LIN {X 70.213, Y 92.532, Z 255.75, A 0, B 90, C 0, E1 0, E2 0, E3 0, E4 0} C_DIS
LIN {X 73.181, Y 90.036, Z 255.75, A 0, B 90, C 0, E1 0, E2 0, E3 0, E4 0} C_DIS
LIN {X 75.725, Y 87.108, Z 255.75, A 0, B 90, C 0, E1 0, E2 0, E3 0, E4 0} C_DIS
LIN {X 77.888, Y 83.886, Z 255.75, A 0, B 90, C 0, E1 0, E2 0, E3 0, E4 0} C_DIS
LIN {X 79.733, Y 80.472, Z 255.75, A 0, B 90, C 0, E1 0, E2 0, E3 0, E4 0} C_DIS
LIN {X 81.33, Y 76.933, Z 255.75, A 0, B 90, C 0, E1 0, E2 0, E3 0, E4 0} C_DIS
LIN {X 82.75, Y 73.32, Z 255.75, A 0, B 90, C 0, E1 0, E2 0, E3 0, E4 0} C_DIS
LIN {X 84.078, Y 69.672, Z 255.75, A 0, B 90, C 0, E1 0, E2 0, E3 0, E4 0} C_DIS
LIN {X 85.426, Y 66.031, Z 255.75, A 0, B 90, C 0, E1 0, E2 0, E3 0, E4 0} C_DIS
LIN {X 86.966, Y 62.469, Z 255.75, A 0, B 90, C 0, E1 0, E2 0, E3 0, E4 0} C_DIS
LIN {X 88.949, Y 59.137, Z 255.75, A 0, B 90, C 0, E1 0, E2 0, E3 0, E4 0} C_DIS
LIN {X 91.538, Y 56.253, Z 255.75, A 0, B 90, C 0, E1 0, E2 0, E3 0, E4 0} C_DIS
LIN {X 94.581, Y 53.847, Z 255.75, A 0, B 90, C 0, E1 0, E2 0, E3 0, E4 0} C_DIS
LIN {X 97.829, Y 51.72, Z 255.75, A 0, B 90, C 0, E1 0, E2 0, E3 0, E4 0} C_DIS
LIN {X 101.131, Y 49.678, Z 255.75, A 0, B 90, C 0, E1 0, E2 0, E3 0, E4 0} C_DIS
LIN {X 104.407, Y 47.594, Z 255.75, A 0, B 90, C 0, E1 0, E2 0, E3 0, E4 0} C_DIS
LIN {X 107.602, Y 45.389, Z 255.75, A 0, B 90, C 0, E1 0, E2 0, E3 0, E4 0} C_DIS
LIN {X 110.666, Y 43.006, Z 255.75, A 0, B 90, C 0, E1 0, E2 0, E3 0, E4 0} C_DIS
LIN {X 113.544, Y 40.402, Z 255.75, A 0, B 90, C 0, E1 0, E2 0, E3 0, E4 0} C_DIS
LIN {X 116.164, Y 37.54, Z 255.75, A 0, B 90, C 0, E1 0, E2 0, E3 0, E4 0} C_DIS
LIN {X 118.433, Y 34.393, Z 255.75, A 0, B 90, C 0, E1 0, E2 0, E3 0, E4 0} C_DIS
LIN {X 120.224, Y 30.953, Z 255.75, A 0, B 90, C 0, E1 0, E2 0, E3 0, E4 0} C_DIS
LIN {X 121.382, Y 27.253, Z 255.75, A 0, B 90, C 0, E1 0, E2 0, E3 0, E4 0} C_DIS
LIN {X 121.779, Y 23.398, Z 255.75, A 0, B 90, C 0, E1 0, E2 0, E3 0, E4 0} C_DIS
LIN {X 121.393, Y 19.541, Z 255.75, A 0, B 90, C 0, E1 0, E2 0, E3 0, E4 0} C_DIS
LIN {X 120.325, Y 15.813, Z 255.75, A 0, B 90, C 0, E1 0, E2 0, E3 0, E4 0} C_DIS
LIN {X 118.73, Y 12.276, Z 255.75, A 0, B 90, C 0, E1 0, E2 0, E3 0, E4 0} C_DIS
LIN {X 116.749, Y 8.94, Z 255.75, A 0, B 90, C 0, E1 0, E2 0, E3 0, E4 0} C_DIS
LIN {X 114.484, Y 5.788, Z 255.75, A 0, B 90, C 0, E1 0, E2 0, E3 0, E4 0} C_DIS
LIN {X 112.003, Y 2.805, Z 255.75, A 0, B 90, C 0, E1 0, E2 0, E3 0, E4 0} C_DIS
LIN {X 109.464, Y 0, Z 255.75, A 0, B 90, C 0, E1 0, E2 0, E3 0, E4 0} C_DIS
LIN {X 106.746, Y -2.436, Z 255.75, A 0, B 90, C 0, E1 0, E2 0, E3 0, E4 0} C_DIS
LIN {X 104.005, Y -5.183, Z 255.75, A 0, B 90, C 0, E1 0, E2 0, E3 0, E4 0} C_DIS
LIN {X 101.28, Y -7.949, Z 255.75, A 0, B 90, C 0, E1 0, E2 0, E3 0, E4 0} C_DIS
LIN {X 98.625, Y -10.781, Z 255.75, A 0, B 90, C 0, E1 0, E2 0, E3 0, E4 0} C_DIS
LIN {X 96.18, Y -13.794, Z 255.75, A 0, B 90, C 0, E1 0, E2 0, E3 0, E4 0} C_DIS
LIN {X 94.209, Y -17.132, Z 255.75, A 0, B 90, C 0, E1 0, E2 0, E3 0, E4 0} C_DIS
LIN {X 93.035, Y -20.823, Z 255.75, A 0, B 90, C 0, E1 0, E2 0, E3 0, E4 0} C_DIS
LIN {X 92.662, Y -24.683, Z 255.75, A 0, B 90, C 0, E1 0, E2 0, E3 0, E4 0} C_DIS
LIN {X 92.802, Y -28.561, Z 255.75, A 0, B 90, C 0, E1 0, E2 0, E3 0, E4 0} C_DIS
LIN {X 93.225, Y -32.42, Z 255.75, A 0, B 90, C 0, E1 0, E2 0, E3 0, E4 0} C_DIS
LIN {X 93.804, Y -36.259, Z 255.75, A 0, B 90, C 0, E1 0, E2 0, E3 0, E4 0} C_DIS
LIN {X 94.463, Y -40.085, Z 255.75, A 0, B 90, C 0, E1 0, E2 0, E3 0, E4 0} C_DIS
LIN {X 95.136, Y -43.908, Z 255.75, A 0, B 90, C 0, E1 0, E2 0, E3 0, E4 0} C_DIS
LIN {X 95.752, Y -47.741, Z 255.75, A 0, B 90, C 0, E1 0, E2 0, E3 0, E4 0} C_DIS
LIN {X 96.227, Y -51.594, Z 255.75, A 0, B 90, C 0, E1 0, E2 0, E3 0, E4 0} C_DIS
LIN {X 96.461, Y -55.469, Z 255.75, A 0, B 90, C 0, E1 0, E2 0, E3 0, E4 0} C_DIS
LIN {X 96.332, Y -59.347, Z 255.75, A 0, B 90, C 0, E1 0, E2 0, E3 0, E4 0} C_DIS
LIN {X 95.702, Y -63.174, Z 255.75, A 0, B 90, C 0, E1 0, E2 0, E3 0, E4 0} C_DIS
LIN {X 94.448, Y -66.843, Z 255.75, A 0, B 90, C 0, E1 0, E2 0, E3 0, E4 0} C_DIS
LIN {X 92.532, Y -70.213, Z 255.75, A 0, B 90, C 0, E1 0, E2 0, E3 0, E4 0} C_DIS
LIN {X 90.036, Y -73.181, Z 255.75, A 0, B 90, C 0, E1 0, E2 0, E3 0, E4 0} C_DIS
LIN {X 87.108, Y -75.725, Z 255.75, A 0, B 90, C 0, E1 0, E2 0, E3 0, E4 0} C_DIS
LIN {X 83.886, Y -77.888, Z 255.75, A 0, B 90, C 0, E1 0, E2 0, E3 0, E4 0} C_DIS
LIN {X 80.472, Y -79.733, Z 255.75, A 0, B 90, C 0, E1 0, E2 0, E3 0, E4 0} C_DIS
LIN {X 76.933, Y -81.33, Z 255.75, A 0, B 90, C 0, E1 0, E2 0, E3 0, E4 0} C_DIS
LIN {X 73.32, Y -82.75, Z 255.75, A 0, B 90, C 0, E1 0, E2 0, E3 0, E4 0} C_DIS
LIN {X 69.672, Y -84.078, Z 255.75, A 0, B 90, C 0, E1 0, E2 0, E3 0, E4 0} C_DIS
LIN {X 66.031, Y -85.426, Z 255.75, A 0, B 90, C 0, E1 0, E2 0, E3 0, E4 0} C_DIS
LIN {X 62.469, Y -86.966, Z 255.75, A 0, B 90, C 0, E1 0, E2 0, E3 0, E4 0} C_DIS
LIN {X 59.137, Y -88.949, Z 255.75, A 0, B 90, C 0, E1 0, E2 0, E3 0, E4 0} C_DIS
LIN {X 56.253, Y -91.538, Z 255.75, A 0, B 90, C 0, E1 0, E2 0, E3 0, E4 0} C_DIS
LIN {X 53.847, Y -94.581, Z 255.75, A 0, B 90, C 0, E1 0, E2 0, E3 0, E4 0} C_DIS
LIN {X 51.72, Y -97.829, Z 255.75, A 0, B 90, C 0, E1 0, E2 0, E3 0, E4 0} C_DIS
LIN {X 49.678, Y -101.131, Z 255.75, A 0, B 90, C 0, E1 0, E2 0, E3 0, E4 0} C_DIS
LIN {X 47.594, Y -104.407, Z 255.75, A 0, B 90, C 0, E1 0, E2 0, E3 0, E4 0} C_DIS
LIN {X 45.389, Y -107.602, Z 255.75, A 0, B 90, C 0, E1 0, E2 0, E3 0, E4 0} C_DIS
LIN {X 43.006, Y -110.666, Z 255.75, A 0, B 90, C 0, E1 0, E2 0, E3 0, E4 0} C_DIS
LIN {X 40.402, Y -113.544, Z 255.75, A 0, B 90, C 0, E1 0, E2 0, E3 0, E4 0} C_DIS
LIN {X 37.54, Y -116.164, Z 255.75, A 0, B 90, C 0, E1 0, E2 0, E3 0, E4 0} C_DIS
LIN {X 34.393, Y -118.433, Z 255.75, A 0, B 90, C 0, E1 0, E2 0, E3 0, E4 0} C_DIS
LIN {X 30.953, Y -120.224, Z 255.75, A 0, B 90, C 0, E1 0, E2 0, E3 0, E4 0} C_DIS
LIN {X 27.253, Y -121.382, Z 255.75, A 0, B 90, C 0, E1 0, E2 0, E3 0, E4 0} C_DIS
LIN {X 23.398, Y -121.779, Z 255.75, A 0, B 90, C 0, E1 0, E2 0, E3 0, E4 0} C_DIS
LIN {X 19.541, Y -121.393, Z 255.75, A 0, B 90, C 0, E1 0, E2 0, E3 0, E4 0} C_DIS
LIN {X 15.813, Y -120.325, Z 255.75, A 0, B 90, C 0, E1 0, E2 0, E3 0, E4 0} C_DIS
LIN {X 12.276, Y -118.73, Z 255.75, A 0, B 90, C 0, E1 0, E2 0, E3 0, E4 0} C_DIS
LIN {X 8.94, Y -116.749, Z 255.75, A 0, B 90, C 0, E1 0, E2 0, E3 0, E4 0} C_DIS
LIN {X 5.788, Y -114.484, Z 255.75, A 0, B 90, C 0, E1 0, E2 0, E3 0, E4 0} C_DIS
LIN {X 2.805, Y -112.003, Z 255.75, A 0, B 90, C 0, E1 0, E2 0, E3 0, E4 0} C_DIS
LIN {X 0, Y -109.464, Z 255.75, A 0, B 90, C 0, E1 0, E2 0, E3 0, E4 0} C_DIS
LIN {X -2.436, Y -106.746, Z 255.75, A 0, B 90, C 0, E1 0, E2 0, E3 0, E4 0} C_DIS
LIN {X -5.183, Y -104.005, Z 255.75, A 0, B 90, C 0, E1 0, E2 0, E3 0, E4 0} C_DIS
LIN {X -7.949, Y -101.28, Z 255.75, A 0, B 90, C 0, E1 0, E2 0, E3 0, E4 0} C_DIS
LIN {X -10.781, Y -98.625, Z 255.75, A 0, B 90, C 0, E1 0, E2 0, E3 0, E4 0} C_DIS
LIN {X -13.794, Y -96.18, Z 255.75, A 0, B 90, C 0, E1 0, E2 0, E3 0, E4 0} C_DIS
LIN {X -17.132, Y -94.209, Z 255.75, A 0, B 90, C 0, E1 0, E2 0, E3 0, E4 0} C_DIS
LIN {X -20.823, Y -93.035, Z 255.75, A 0, B 90, C 0, E1 0, E2 0, E3 0, E4 0} C_DIS
LIN {X -24.683, Y -92.662, Z 255.75, A 0, B 90, C 0, E1 0, E2 0, E3 0, E4 0} C_DIS
LIN {X -28.561, Y -92.802, Z 255.75, A 0, B 90, C 0, E1 0, E2 0, E3 0, E4 0} C_DIS
LIN {X -32.42, Y -93.225, Z 255.75, A 0, B 90, C 0, E1 0, E2 0, E3 0, E4 0} C_DIS
LIN {X -36.259, Y -93.804, Z 255.75, A 0, B 90, C 0, E1 0, E2 0, E3 0, E4 0} C_DIS
LIN {X -40.085, Y -94.463, Z 255.75, A 0, B 90, C 0, E1 0, E2 0, E3 0, E4 0} C_DIS
LIN {X -43.908, Y -95.136, Z 255.75, A 0, B 90, C 0, E1 0, E2 0, E3 0, E4 0} C_DIS
LIN {X -47.741, Y -95.752, Z 255.75, A 0, B 90, C 0, E1 0, E2 0, E3 0, E4 0} C_DIS
LIN {X -51.594, Y -96.227, Z 255.75, A 0, B 90, C 0, E1 0, E2 0, E3 0, E4 0} C_DIS
LIN {X -55.469, Y -96.461, Z 255.75, A 0, B 90, C 0, E1 0, E2 0, E3 0, E4 0} C_DIS
LIN {X -59.347, Y -96.332, Z 255.75, A 0, B 90, C 0, E1 0, E2 0, E3 0, E4 0} C_DIS
LIN {X -63.174, Y -95.702, Z 255.75, A 0, B 90, C 0, E1 0, E2 0, E3 0, E4 0} C_DIS
LIN {X -66.843, Y -94.448, Z 255.75, A 0, B 90, C 0, E1 0, E2 0, E3 0, E4 0} C_DIS
LIN {X -70.213, Y -92.532, Z 255.75, A 0, B 90, C 0, E1 0, E2 0, E3 0, E4 0} C_DIS
LIN {X -73.181, Y -90.036, Z 255.75, A 0, B 90, C 0, E1 0, E2 0, E3 0, E4 0} C_DIS
LIN {X -75.725, Y -87.108, Z 255.75, A 0, B 90, C 0, E1 0, E2 0, E3 0, E4 0} C_DIS
LIN {X -77.888, Y -83.886, Z 255.75, A 0, B 90, C 0, E1 0, E2 0, E3 0, E4 0} C_DIS
LIN {X -79.733, Y -80.472, Z 255.75, A 0, B 90, C 0, E1 0, E2 0, E3 0, E4 0} C_DIS
LIN {X -81.33, Y -76.933, Z 255.75, A 0, B 90, C 0, E1 0, E2 0, E3 0, E4 0} C_DIS
LIN {X -82.75, Y -73.32, Z 255.75, A 0, B 90, C 0, E1 0, E2 0, E3 0, E4 0} C_DIS
LIN {X -84.078, Y -69.672, Z 255.75, A 0, B 90, C 0, E1 0, E2 0, E3 0, E4 0} C_DIS
LIN {X -85.426, Y -66.031, Z 255.75, A 0, B 90, C 0, E1 0, E2 0, E3 0, E4 0} C_DIS
LIN {X -86.966, Y -62.469, Z 255.75, A 0, B 90, C 0, E1 0, E2 0, E3 0, E4 0} C_DIS
LIN {X -88.949, Y -59.137, Z 255.75, A 0, B 90, C 0, E1 0, E2 0, E3 0, E4 0} C_DIS
LIN {X -91.538, Y -56.253, Z 255.75, A 0, B 90, C 0, E1 0, E2 0, E3 0, E4 0} C_DIS
LIN {X -94.581, Y -53.847, Z 255.75, A 0, B 90, C 0, E1 0, E2 0, E3 0, E4 0} C_DIS
LIN {X -97.829, Y -51.72, Z 255.75, A 0, B 90, C 0, E1 0, E2 0, E3 0, E4 0} C_DIS
LIN {X -101.131, Y -49.678, Z 255.75, A 0, B 90, C 0, E1 0, E2 0, E3 0, E4 0} C_DIS
LIN {X -104.407, Y -47.594, Z 255.75, A 0, B 90, C 0, E1 0, E2 0, E3 0, E4 0} C_DIS
LIN {X -107.602, Y -45.389, Z 255.75, A 0, B 90, C 0, E1 0, E2 0, E3 0, E4 0} C_DIS
LIN {X -110.666, Y -43.006, Z 255.75, A 0, B 90, C 0, E1 0, E2 0, E3 0, E4 0} C_DIS
LIN {X -113.544, Y -40.402, Z 255.75, A 0, B 90, C 0, E1 0, E2 0, E3 0, E4 0} C_DIS
LIN {X -116.164, Y -37.54, Z 255.75, A 0, B 90, C 0, E1 0, E2 0, E3 0, E4 0} C_DIS
LIN {X -118.433, Y -34.393, Z 255.75, A 0, B 90, C 0, E1 0, E2 0, E3 0, E4 0} C_DIS
LIN {X -120.224, Y -30.953, Z 255.75, A 0, B 90, C 0, E1 0, E2 0, E3 0, E4 0} C_DIS
LIN {X -121.382, Y -27.253, Z 255.75, A 0, B 90, C 0, E1 0, E2 0, E3 0, E4 0} C_DIS
LIN {X -121.779, Y -23.398, Z 255.75, A 0, B 90, C 0, E1 0, E2 0, E3 0, E4 0} C_DIS
LIN {X -121.393, Y -19.541, Z 255.75, A 0, B 90, C 0, E1 0, E2 0, E3 0, E4 0} C_DIS
LIN {X -120.325, Y -15.813, Z 255.75, A 0, B 90, C 0, E1 0, E2 0, E3 0, E4 0} C_DIS
LIN {X -118.73, Y -12.276, Z 255.75, A 0, B 90, C 0, E1 0, E2 0, E3 0, E4 0} C_DIS
LIN {X -116.749, Y -8.94, Z 255.75, A 0, B 90, C 0, E1 0, E2 0, E3 0, E4 0} C_DIS
LIN {X -114.484, Y -5.788, Z 255.75, A 0, B 90, C 0, E1 0, E2 0, E3 0, E4 0} C_DIS
LIN {X -112.003, Y -2.805, Z 255.75, A 0, B 90, C 0, E1 0, E2 0, E3 0, E4 0} C_DIS
LIN {X -110.257, Y 0, Z 258.25, A 0, B 90, C 0, E1 0, E2 0, E3 0, E4 0} C_DIS
LIN {X -107.504, Y 2.463, Z 258.25, A 0, B 90, C 0, E1 0, E2 0, E3 0, E4 0} C_DIS
LIN {X -104.727, Y 5.233, Z 258.25, A 0, B 90, C 0, E1 0, E2 0, E3 0, E4 0} C_DIS
LIN {X -101.968, Y 8.022, Z 258.25, A 0, B 90, C 0, E1 0, E2 0, E3 0, E4 0} C_DIS
LIN {X -99.284, Y 10.883, Z 258.25, A 0, B 90, C 0, E1 0, E2 0, E3 0, E4 0} C_DIS
LIN {X -96.821, Y 13.934, Z 258.25, A 0, B 90, C 0, E1 0, E2 0, E3 0, E4 0} C_DIS
LIN {X -94.856, Y 17.323, Z 258.25, A 0, B 90, C 0, E1 0, E2 0, E3 0, E4 0} C_DIS
LIN {X -93.725, Y 21.069, Z 258.25, A 0, B 90, C 0, E1 0, E2 0, E3 0, E4 0} C_DIS
LIN {X -93.423, Y 24.976, Z 258.25, A 0, B 90, C 0, E1 0, E2 0, E3 0, E4 0} C_DIS
LIN {X -93.644, Y 28.891, Z 258.25, A 0, B 90, C 0, E1 0, E2 0, E3 0, E4 0} C_DIS
LIN {X -94.147, Y 32.782, Z 258.25, A 0, B 90, C 0, E1 0, E2 0, E3 0, E4 0} C_DIS
LIN {X -94.799, Y 36.651, Z 258.25, A 0, B 90, C 0, E1 0, E2 0, E3 0, E4 0} C_DIS
LIN {X -95.522, Y 40.507, Z 258.25, A 0, B 90, C 0, E1 0, E2 0, E3 0, E4 0} C_DIS
LIN {X -96.247, Y 44.362, Z 258.25, A 0, B 90, C 0, E1 0, E2 0, E3 0, E4 0} C_DIS
LIN {X -96.904, Y 48.23, Z 258.25, A 0, B 90, C 0, E1 0, E2 0, E3 0, E4 0} C_DIS
LIN {X -97.406, Y 52.121, Z 258.25, A 0, B 90, C 0, E1 0, E2 0, E3 0, E4 0} C_DIS
LIN {X -97.652, Y 56.036, Z 258.25, A 0, B 90, C 0, E1 0, E2 0, E3 0, E4 0} C_DIS
LIN {X -97.516, Y 59.954, Z 258.25, A 0, B 90, C 0, E1 0, E2 0, E3 0, E4 0} C_DIS
LIN {X -96.856, Y 63.818, Z 258.25, A 0, B 90, C 0, E1 0, E2 0, E3 0, E4 0} C_DIS
LIN {X -95.547, Y 67.51, Z 258.25, A 0, B 90, C 0, E1 0, E2 0, E3 0, E4 0} C_DIS
LIN {X -93.554, Y 70.883, Z 258.25, A 0, B 90, C 0, E1 0, E2 0, E3 0, E4 0} C_DIS
LIN {X -90.97, Y 73.828, Z 258.25, A 0, B 90, C 0, E1 0, E2 0, E3 0, E4 0} C_DIS
LIN {X -87.951, Y 76.329, Z 258.25, A 0, B 90, C 0, E1 0, E2 0, E3 0, E4 0} C_DIS
LIN {X -84.641, Y 78.43, Z 258.25, A 0, B 90, C 0, E1 0, E2 0, E3 0, E4 0} C_DIS
LIN {X -81.142, Y 80.203, Z 258.25, A 0, B 90, C 0, E1 0, E2 0, E3 0, E4 0} C_DIS
LIN {X -77.525, Y 81.722, Z 258.25, A 0, B 90, C 0, E1 0, E2 0, E3 0, E4 0} C_DIS
LIN {X -73.838, Y 83.062, Z 258.25, A 0, B 90, C 0, E1 0, E2 0, E3 0, E4 0} C_DIS
LIN {X -70.12, Y 84.313, Z 258.25, A 0, B 90, C 0, E1 0, E2 0, E3 0, E4 0} C_DIS
LIN {X -66.41, Y 85.591, Z 258.25, A 0, B 90, C 0, E1 0, E2 0, E3 0, E4 0} C_DIS
LIN {X -62.78, Y 87.076, Z 258.25, A 0, B 90, C 0, E1 0, E2 0, E3 0, E4 0} C_DIS
LIN {X -59.382, Y 89.026, Z 258.25, A 0, B 90, C 0, E1 0, E2 0, E3 0, E4 0} C_DIS
LIN {X -56.445, Y 91.617, Z 258.25, A 0, B 90, C 0, E1 0, E2 0, E3 0, E4 0} C_DIS
LIN {X -54.013, Y 94.691, Z 258.25, A 0, B 90, C 0, E1 0, E2 0, E3 0, E4 0} C_DIS
LIN {X -51.883, Y 97.985, Z 258.25, A 0, B 90, C 0, E1 0, E2 0, E3 0, E4 0} C_DIS
LIN {X -49.852, Y 101.342, Z 258.25, A 0, B 90, C 0, E1 0, E2 0, E3 0, E4 0} C_DIS
LIN {X -47.788, Y 104.679, Z 258.25, A 0, B 90, C 0, E1 0, E2 0, E3 0, E4 0} C_DIS
LIN {X -45.608, Y 107.94, Z 258.25, A 0, B 90, C 0, E1 0, E2 0, E3 0, E4 0} C_DIS
LIN {X -43.252, Y 111.076, Z 258.25, A 0, B 90, C 0, E1 0, E2 0, E3 0, E4 0} C_DIS
LIN {X -40.673, Y 114.031, Z 258.25, A 0, B 90, C 0, E1 0, E2 0, E3 0, E4 0} C_DIS
LIN {X -37.831, Y 116.734, Z 258.25, A 0, B 90, C 0, E1 0, E2 0, E3 0, E4 0} C_DIS
LIN {X -34.696, Y 119.088, Z 258.25, A 0, B 90, C 0, E1 0, E2 0, E3 0, E4 0} C_DIS
LIN {X -31.254, Y 120.962, Z 258.25, A 0, B 90, C 0, E1 0, E2 0, E3 0, E4 0} C_DIS
LIN {X -27.536, Y 122.195, Z 258.25, A 0, B 90, C 0, E1 0, E2 0, E3 0, E4 0} C_DIS
LIN {X -23.646, Y 122.65, Z 258.25, A 0, B 90, C 0, E1 0, E2 0, E3 0, E4 0} C_DIS
LIN {X -19.745, Y 122.297, Z 258.25, A 0, B 90, C 0, E1 0, E2 0, E3 0, E4 0} C_DIS
LIN {X -15.972, Y 121.239, Z 258.25, A 0, B 90, C 0, E1 0, E2 0, E3 0, E4 0} C_DIS
LIN {X -12.394, Y 119.636, Z 258.25, A 0, B 90, C 0, E1 0, E2 0, E3 0, E4 0} C_DIS
LIN {X -9.021, Y 117.635, Z 258.25, A 0, B 90, C 0, E1 0, E2 0, E3 0, E4 0} C_DIS
LIN {X -5.839, Y 115.342, Z 258.25, A 0, B 90, C 0, E1 0, E2 0, E3 0, E4 0} C_DIS
LIN {X -2.829, Y 112.83, Z 258.25, A 0, B 90, C 0, E1 0, E2 0, E3 0, E4 0} C_DIS
LIN {X 0, Y 110.257, Z 258.25, A 0, B 90, C 0, E1 0, E2 0, E3 0, E4 0} C_DIS
LIN {X 2.463, Y 107.504, Z 258.25, A 0, B 90, C 0, E1 0, E2 0, E3 0, E4 0} C_DIS
LIN {X 5.233, Y 104.727, Z 258.25, A 0, B 90, C 0, E1 0, E2 0, E3 0, E4 0} C_DIS
LIN {X 8.022, Y 101.968, Z 258.25, A 0, B 90, C 0, E1 0, E2 0, E3 0, E4 0} C_DIS
LIN {X 10.883, Y 99.284, Z 258.25, A 0, B 90, C 0, E1 0, E2 0, E3 0, E4 0} C_DIS
LIN {X 13.934, Y 96.821, Z 258.25, A 0, B 90, C 0, E1 0, E2 0, E3 0, E4 0} C_DIS
LIN {X 17.323, Y 94.856, Z 258.25, A 0, B 90, C 0, E1 0, E2 0, E3 0, E4 0} C_DIS
LIN {X 21.069, Y 93.725, Z 258.25, A 0, B 90, C 0, E1 0, E2 0, E3 0, E4 0} C_DIS
LIN {X 24.976, Y 93.423, Z 258.25, A 0, B 90, C 0, E1 0, E2 0, E3 0, E4 0} C_DIS
LIN {X 28.891, Y 93.644, Z 258.25, A 0, B 90, C 0, E1 0, E2 0, E3 0, E4 0} C_DIS
LIN {X 32.782, Y 94.147, Z 258.25, A 0, B 90, C 0, E1 0, E2 0, E3 0, E4 0} C_DIS
LIN {X 36.651, Y 94.799, Z 258.25, A 0, B 90, C 0, E1 0, E2 0, E3 0, E4 0} C_DIS
LIN {X 40.507, Y 95.522, Z 258.25, A 0, B 90, C 0, E1 0, E2 0, E3 0, E4 0} C_DIS
LIN {X 44.362, Y 96.247, Z 258.25, A 0, B 90, C 0, E1 0, E2 0, E3 0, E4 0} C_DIS
LIN {X 48.23, Y 96.904, Z 258.25, A 0, B 90, C 0, E1 0, E2 0, E3 0, E4 0} C_DIS
LIN {X 52.121, Y 97.406, Z 258.25, A 0, B 90, C 0, E1 0, E2 0, E3 0, E4 0} C_DIS
LIN {X 56.036, Y 97.652, Z 258.25, A 0, B 90, C 0, E1 0, E2 0, E3 0, E4 0} C_DIS
LIN {X 59.954, Y 97.516, Z 258.25, A 0, B 90, C 0, E1 0, E2 0, E3 0, E4 0} C_DIS
LIN {X 63.818, Y 96.856, Z 258.25, A 0, B 90, C 0, E1 0, E2 0, E3 0, E4 0} C_DIS
LIN {X 67.51, Y 95.547, Z 258.25, A 0, B 90, C 0, E1 0, E2 0, E3 0, E4 0} C_DIS
LIN {X 70.883, Y 93.554, Z 258.25, A 0, B 90, C 0, E1 0, E2 0, E3 0, E4 0} C_DIS
LIN {X 73.828, Y 90.97, Z 258.25, A 0, B 90, C 0, E1 0, E2 0, E3 0, E4 0} C_DIS
LIN {X 76.329, Y 87.951, Z 258.25, A 0, B 90, C 0, E1 0, E2 0, E3 0, E4 0} C_DIS
LIN {X 78.43, Y 84.641, Z 258.25, A 0, B 90, C 0, E1 0, E2 0, E3 0, E4 0} C_DIS
LIN {X 80.203, Y 81.142, Z 258.25, A 0, B 90, C 0, E1 0, E2 0, E3 0, E4 0} C_DIS
LIN {X 81.722, Y 77.525, Z 258.25, A 0, B 90, C 0, E1 0, E2 0, E3 0, E4 0} C_DIS
LIN {X 83.062, Y 73.838, Z 258.25, A 0, B 90, C 0, E1 0, E2 0, E3 0, E4 0} C_DIS
LIN {X 84.313, Y 70.12, Z 258.25, A 0, B 90, C 0, E1 0, E2 0, E3 0, E4 0} C_DIS
LIN {X 85.591, Y 66.41, Z 258.25, A 0, B 90, C 0, E1 0, E2 0, E3 0, E4 0} C_DIS
LIN {X 87.076, Y 62.78, Z 258.25, A 0, B 90, C 0, E1 0, E2 0, E3 0, E4 0} C_DIS
LIN {X 89.026, Y 59.382, Z 258.25, A 0, B 90, C 0, E1 0, E2 0, E3 0, E4 0} C_DIS
LIN {X 91.617, Y 56.445, Z 258.25, A 0, B 90, C 0, E1 0, E2 0, E3 0, E4 0} C_DIS
LIN {X 94.691, Y 54.013, Z 258.25, A 0, B 90, C 0, E1 0, E2 0, E3 0, E4 0} C_DIS
LIN {X 97.985, Y 51.883, Z 258.25, A 0, B 90, C 0, E1 0, E2 0, E3 0, E4 0} C_DIS
LIN {X 101.342, Y 49.852, Z 258.25, A 0, B 90, C 0, E1 0, E2 0, E3 0, E4 0} C_DIS
LIN {X 104.679, Y 47.788, Z 258.25, A 0, B 90, C 0, E1 0, E2 0, E3 0, E4 0} C_DIS
LIN {X 107.94, Y 45.608, Z 258.25, A 0, B 90, C 0, E1 0, E2 0, E3 0, E4 0} C_DIS
LIN {X 111.076, Y 43.252, Z 258.25, A 0, B 90, C 0, E1 0, E2 0, E3 0, E4 0} C_DIS
LIN {X 114.031, Y 40.673, Z 258.25, A 0, B 90, C 0, E1 0, E2 0, E3 0, E4 0} C_DIS
LIN {X 116.734, Y 37.831, Z 258.25, A 0, B 90, C 0, E1 0, E2 0, E3 0, E4 0} C_DIS
LIN {X 119.088, Y 34.696, Z 258.25, A 0, B 90, C 0, E1 0, E2 0, E3 0, E4 0} C_DIS
LIN {X 120.962, Y 31.254, Z 258.25, A 0, B 90, C 0, E1 0, E2 0, E3 0, E4 0} C_DIS
LIN {X 122.195, Y 27.536, Z 258.25, A 0, B 90, C 0, E1 0, E2 0, E3 0, E4 0} C_DIS
LIN {X 122.65, Y 23.646, Z 258.25, A 0, B 90, C 0, E1 0, E2 0, E3 0, E4 0} C_DIS
LIN {X 122.297, Y 19.745, Z 258.25, A 0, B 90, C 0, E1 0, E2 0, E3 0, E4 0} C_DIS
LIN {X 121.239, Y 15.972, Z 258.25, A 0, B 90, C 0, E1 0, E2 0, E3 0, E4 0} C_DIS
LIN {X 119.636, Y 12.394, Z 258.25, A 0, B 90, C 0, E1 0, E2 0, E3 0, E4 0} C_DIS
LIN {X 117.635, Y 9.021, Z 258.25, A 0, B 90, C 0, E1 0, E2 0, E3 0, E4 0} C_DIS
LIN {X 115.342, Y 5.839, Z 258.25, A 0, B 90, C 0, E1 0, E2 0, E3 0, E4 0} C_DIS
LIN {X 112.83, Y 2.829, Z 258.25, A 0, B 90, C 0, E1 0, E2 0, E3 0, E4 0} C_DIS
LIN {X 110.257, Y 0, Z 258.25, A 0, B 90, C 0, E1 0, E2 0, E3 0, E4 0} C_DIS
LIN {X 107.504, Y -2.463, Z 258.25, A 0, B 90, C 0, E1 0, E2 0, E3 0, E4 0} C_DIS
LIN {X 104.727, Y -5.233, Z 258.25, A 0, B 90, C 0, E1 0, E2 0, E3 0, E4 0} C_DIS
LIN {X 101.968, Y -8.022, Z 258.25, A 0, B 90, C 0, E1 0, E2 0, E3 0, E4 0} C_DIS
LIN {X 99.284, Y -10.883, Z 258.25, A 0, B 90, C 0, E1 0, E2 0, E3 0, E4 0} C_DIS
LIN {X 96.821, Y -13.934, Z 258.25, A 0, B 90, C 0, E1 0, E2 0, E3 0, E4 0} C_DIS
LIN {X 94.856, Y -17.323, Z 258.25, A 0, B 90, C 0, E1 0, E2 0, E3 0, E4 0} C_DIS
LIN {X 93.725, Y -21.069, Z 258.25, A 0, B 90, C 0, E1 0, E2 0, E3 0, E4 0} C_DIS
LIN {X 93.423, Y -24.976, Z 258.25, A 0, B 90, C 0, E1 0, E2 0, E3 0, E4 0} C_DIS
LIN {X 93.644, Y -28.891, Z 258.25, A 0, B 90, C 0, E1 0, E2 0, E3 0, E4 0} C_DIS
LIN {X 94.147, Y -32.782, Z 258.25, A 0, B 90, C 0, E1 0, E2 0, E3 0, E4 0} C_DIS
LIN {X 94.799, Y -36.651, Z 258.25, A 0, B 90, C 0, E1 0, E2 0, E3 0, E4 0} C_DIS
LIN {X 95.522, Y -40.507, Z 258.25, A 0, B 90, C 0, E1 0, E2 0, E3 0, E4 0} C_DIS
LIN {X 96.247, Y -44.362, Z 258.25, A 0, B 90, C 0, E1 0, E2 0, E3 0, E4 0} C_DIS
LIN {X 96.904, Y -48.23, Z 258.25, A 0, B 90, C 0, E1 0, E2 0, E3 0, E4 0} C_DIS
LIN {X 97.406, Y -52.121, Z 258.25, A 0, B 90, C 0, E1 0, E2 0, E3 0, E4 0} C_DIS
LIN {X 97.652, Y -56.036, Z 258.25, A 0, B 90, C 0, E1 0, E2 0, E3 0, E4 0} C_DIS
LIN {X 97.516, Y -59.954, Z 258.25, A 0, B 90, C 0, E1 0, E2 0, E3 0, E4 0} C_DIS
LIN {X 96.856, Y -63.818, Z 258.25, A 0, B 90, C 0, E1 0, E2 0, E3 0, E4 0} C_DIS
LIN {X 95.547, Y -67.51, Z 258.25, A 0, B 90, C 0, E1 0, E2 0, E3 0, E4 0} C_DIS
LIN {X 93.554, Y -70.883, Z 258.25, A 0, B 90, C 0, E1 0, E2 0, E3 0, E4 0} C_DIS
LIN {X 90.97, Y -73.828, Z 258.25, A 0, B 90, C 0, E1 0, E2 0, E3 0, E4 0} C_DIS
LIN {X 87.951, Y -76.329, Z 258.25, A 0, B 90, C 0, E1 0, E2 0, E3 0, E4 0} C_DIS
LIN {X 84.641, Y -78.43, Z 258.25, A 0, B 90, C 0, E1 0, E2 0, E3 0, E4 0} C_DIS
LIN {X 81.142, Y -80.203, Z 258.25, A 0, B 90, C 0, E1 0, E2 0, E3 0, E4 0} C_DIS
LIN {X 77.525, Y -81.722, Z 258.25, A 0, B 90, C 0, E1 0, E2 0, E3 0, E4 0} C_DIS
LIN {X 73.838, Y -83.062, Z 258.25, A 0, B 90, C 0, E1 0, E2 0, E3 0, E4 0} C_DIS
LIN {X 70.12, Y -84.313, Z 258.25, A 0, B 90, C 0, E1 0, E2 0, E3 0, E4 0} C_DIS
LIN {X 66.41, Y -85.591, Z 258.25, A 0, B 90, C 0, E1 0, E2 0, E3 0, E4 0} C_DIS
LIN {X 62.78, Y -87.076, Z 258.25, A 0, B 90, C 0, E1 0, E2 0, E3 0, E4 0} C_DIS
LIN {X 59.382, Y -89.026, Z 258.25, A 0, B 90, C 0, E1 0, E2 0, E3 0, E4 0} C_DIS
LIN {X 56.445, Y -91.617, Z 258.25, A 0, B 90, C 0, E1 0, E2 0, E3 0, E4 0} C_DIS
LIN {X 54.013, Y -94.691, Z 258.25, A 0, B 90, C 0, E1 0, E2 0, E3 0, E4 0} C_DIS
LIN {X 51.883, Y -97.985, Z 258.25, A 0, B 90, C 0, E1 0, E2 0, E3 0, E4 0} C_DIS
LIN {X 49.852, Y -101.342, Z 258.25, A 0, B 90, C 0, E1 0, E2 0, E3 0, E4 0} C_DIS
LIN {X 47.788, Y -104.679, Z 258.25, A 0, B 90, C 0, E1 0, E2 0, E3 0, E4 0} C_DIS
LIN {X 45.608, Y -107.94, Z 258.25, A 0, B 90, C 0, E1 0, E2 0, E3 0, E4 0} C_DIS
LIN {X 43.252, Y -111.076, Z 258.25, A 0, B 90, C 0, E1 0, E2 0, E3 0, E4 0} C_DIS
LIN {X 40.673, Y -114.031, Z 258.25, A 0, B 90, C 0, E1 0, E2 0, E3 0, E4 0} C_DIS
LIN {X 37.831, Y -116.734, Z 258.25, A 0, B 90, C 0, E1 0, E2 0, E3 0, E4 0} C_DIS
LIN {X 34.696, Y -119.088, Z 258.25, A 0, B 90, C 0, E1 0, E2 0, E3 0, E4 0} C_DIS
LIN {X 31.254, Y -120.962, Z 258.25, A 0, B 90, C 0, E1 0, E2 0, E3 0, E4 0} C_DIS
LIN {X 27.536, Y -122.195, Z 258.25, A 0, B 90, C 0, E1 0, E2 0, E3 0, E4 0} C_DIS
LIN {X 23.646, Y -122.65, Z 258.25, A 0, B 90, C 0, E1 0, E2 0, E3 0, E4 0} C_DIS
LIN {X 19.745, Y -122.297, Z 258.25, A 0, B 90, C 0, E1 0, E2 0, E3 0, E4 0} C_DIS
LIN {X 15.972, Y -121.239, Z 258.25, A 0, B 90, C 0, E1 0, E2 0, E3 0, E4 0} C_DIS
LIN {X 12.394, Y -119.636, Z 258.25, A 0, B 90, C 0, E1 0, E2 0, E3 0, E4 0} C_DIS
LIN {X 9.021, Y -117.635, Z 258.25, A 0, B 90, C 0, E1 0, E2 0, E3 0, E4 0} C_DIS
LIN {X 5.839, Y -115.342, Z 258.25, A 0, B 90, C 0, E1 0, E2 0, E3 0, E4 0} C_DIS
LIN {X 2.829, Y -112.83, Z 258.25, A 0, B 90, C 0, E1 0, E2 0, E3 0, E4 0} C_DIS
LIN {X 0, Y -110.257, Z 258.25, A 0, B 90, C 0, E1 0, E2 0, E3 0, E4 0} C_DIS
LIN {X -2.463, Y -107.504, Z 258.25, A 0, B 90, C 0, E1 0, E2 0, E3 0, E4 0} C_DIS
LIN {X -5.233, Y -104.727, Z 258.25, A 0, B 90, C 0, E1 0, E2 0, E3 0, E4 0} C_DIS
LIN {X -8.022, Y -101.968, Z 258.25, A 0, B 90, C 0, E1 0, E2 0, E3 0, E4 0} C_DIS
LIN {X -10.883, Y -99.284, Z 258.25, A 0, B 90, C 0, E1 0, E2 0, E3 0, E4 0} C_DIS
LIN {X -13.934, Y -96.821, Z 258.25, A 0, B 90, C 0, E1 0, E2 0, E3 0, E4 0} C_DIS
LIN {X -17.323, Y -94.856, Z 258.25, A 0, B 90, C 0, E1 0, E2 0, E3 0, E4 0} C_DIS
LIN {X -21.069, Y -93.725, Z 258.25, A 0, B 90, C 0, E1 0, E2 0, E3 0, E4 0} C_DIS
LIN {X -24.976, Y -93.423, Z 258.25, A 0, B 90, C 0, E1 0, E2 0, E3 0, E4 0} C_DIS
LIN {X -28.891, Y -93.644, Z 258.25, A 0, B 90, C 0, E1 0, E2 0, E3 0, E4 0} C_DIS
LIN {X -32.782, Y -94.147, Z 258.25, A 0, B 90, C 0, E1 0, E2 0, E3 0, E4 0} C_DIS
LIN {X -36.651, Y -94.799, Z 258.25, A 0, B 90, C 0, E1 0, E2 0, E3 0, E4 0} C_DIS
LIN {X -40.507, Y -95.522, Z 258.25, A 0, B 90, C 0, E1 0, E2 0, E3 0, E4 0} C_DIS
LIN {X -44.362, Y -96.247, Z 258.25, A 0, B 90, C 0, E1 0, E2 0, E3 0, E4 0} C_DIS
LIN {X -48.23, Y -96.904, Z 258.25, A 0, B 90, C 0, E1 0, E2 0, E3 0, E4 0} C_DIS
LIN {X -52.121, Y -97.406, Z 258.25, A 0, B 90, C 0, E1 0, E2 0, E3 0, E4 0} C_DIS
LIN {X -56.036, Y -97.652, Z 258.25, A 0, B 90, C 0, E1 0, E2 0, E3 0, E4 0} C_DIS
LIN {X -59.954, Y -97.516, Z 258.25, A 0, B 90, C 0, E1 0, E2 0, E3 0, E4 0} C_DIS
LIN {X -63.818, Y -96.856, Z 258.25, A 0, B 90, C 0, E1 0, E2 0, E3 0, E4 0} C_DIS
LIN {X -67.51, Y -95.547, Z 258.25, A 0, B 90, C 0, E1 0, E2 0, E3 0, E4 0} C_DIS
LIN {X -70.883, Y -93.554, Z 258.25, A 0, B 90, C 0, E1 0, E2 0, E3 0, E4 0} C_DIS
LIN {X -73.828, Y -90.97, Z 258.25, A 0, B 90, C 0, E1 0, E2 0, E3 0, E4 0} C_DIS
LIN {X -76.329, Y -87.951, Z 258.25, A 0, B 90, C 0, E1 0, E2 0, E3 0, E4 0} C_DIS
LIN {X -78.43, Y -84.641, Z 258.25, A 0, B 90, C 0, E1 0, E2 0, E3 0, E4 0} C_DIS
LIN {X -80.203, Y -81.142, Z 258.25, A 0, B 90, C 0, E1 0, E2 0, E3 0, E4 0} C_DIS
LIN {X -81.722, Y -77.525, Z 258.25, A 0, B 90, C 0, E1 0, E2 0, E3 0, E4 0} C_DIS
LIN {X -83.062, Y -73.838, Z 258.25, A 0, B 90, C 0, E1 0, E2 0, E3 0, E4 0} C_DIS
LIN {X -84.313, Y -70.12, Z 258.25, A 0, B 90, C 0, E1 0, E2 0, E3 0, E4 0} C_DIS
LIN {X -85.591, Y -66.41, Z 258.25, A 0, B 90, C 0, E1 0, E2 0, E3 0, E4 0} C_DIS
LIN {X -87.076, Y -62.78, Z 258.25, A 0, B 90, C 0, E1 0, E2 0, E3 0, E4 0} C_DIS
LIN {X -89.026, Y -59.382, Z 258.25, A 0, B 90, C 0, E1 0, E2 0, E3 0, E4 0} C_DIS
LIN {X -91.617, Y -56.445, Z 258.25, A 0, B 90, C 0, E1 0, E2 0, E3 0, E4 0} C_DIS
LIN {X -94.691, Y -54.013, Z 258.25, A 0, B 90, C 0, E1 0, E2 0, E3 0, E4 0} C_DIS
LIN {X -97.985, Y -51.883, Z 258.25, A 0, B 90, C 0, E1 0, E2 0, E3 0, E4 0} C_DIS
LIN {X -101.342, Y -49.852, Z 258.25, A 0, B 90, C 0, E1 0, E2 0, E3 0, E4 0} C_DIS
LIN {X -104.679, Y -47.788, Z 258.25, A 0, B 90, C 0, E1 0, E2 0, E3 0, E4 0} C_DIS
LIN {X -107.94, Y -45.608, Z 258.25, A 0, B 90, C 0, E1 0, E2 0, E3 0, E4 0} C_DIS
LIN {X -111.076, Y -43.252, Z 258.25, A 0, B 90, C 0, E1 0, E2 0, E3 0, E4 0} C_DIS
LIN {X -114.031, Y -40.673, Z 258.25, A 0, B 90, C 0, E1 0, E2 0, E3 0, E4 0} C_DIS
LIN {X -116.734, Y -37.831, Z 258.25, A 0, B 90, C 0, E1 0, E2 0, E3 0, E4 0} C_DIS
LIN {X -119.088, Y -34.696, Z 258.25, A 0, B 90, C 0, E1 0, E2 0, E3 0, E4 0} C_DIS
LIN {X -120.962, Y -31.254, Z 258.25, A 0, B 90, C 0, E1 0, E2 0, E3 0, E4 0} C_DIS
LIN {X -122.195, Y -27.536, Z 258.25, A 0, B 90, C 0, E1 0, E2 0, E3 0, E4 0} C_DIS
LIN {X -122.65, Y -23.646, Z 258.25, A 0, B 90, C 0, E1 0, E2 0, E3 0, E4 0} C_DIS
LIN {X -122.297, Y -19.745, Z 258.25, A 0, B 90, C 0, E1 0, E2 0, E3 0, E4 0} C_DIS
LIN {X -121.239, Y -15.972, Z 258.25, A 0, B 90, C 0, E1 0, E2 0, E3 0, E4 0} C_DIS
LIN {X -119.636, Y -12.394, Z 258.25, A 0, B 90, C 0, E1 0, E2 0, E3 0, E4 0} C_DIS
LIN {X -117.635, Y -9.021, Z 258.25, A 0, B 90, C 0, E1 0, E2 0, E3 0, E4 0} C_DIS
LIN {X -115.342, Y -5.839, Z 258.25, A 0, B 90, C 0, E1 0, E2 0, E3 0, E4 0} C_DIS
LIN {X -112.83, Y -2.829, Z 258.25, A 0, B 90, C 0, E1 0, E2 0, E3 0, E4 0} C_DIS
LIN {X -111.06, Y 0, Z 260.75, A 0, B 90, C 0, E1 0, E2 0, E3 0, E4 0} C_DIS
LIN {X -108.272, Y 2.491, Z 260.75, A 0, B 90, C 0, E1 0, E2 0, E3 0, E4 0} C_DIS
LIN {X -105.459, Y 5.284, Z 260.75, A 0, B 90, C 0, E1 0, E2 0, E3 0, E4 0} C_DIS
LIN {X -102.664, Y 8.097, Z 260.75, A 0, B 90, C 0, E1 0, E2 0, E3 0, E4 0} C_DIS
LIN {X -99.951, Y 10.989, Z 260.75, A 0, B 90, C 0, E1 0, E2 0, E3 0, E4 0} C_DIS
LIN {X -97.469, Y 14.079, Z 260.75, A 0, B 90, C 0, E1 0, E2 0, E3 0, E4 0} C_DIS
LIN {X -95.512, Y 17.52, Z 260.75, A 0, B 90, C 0, E1 0, E2 0, E3 0, E4 0} C_DIS
LIN {X -94.427, Y 21.323, Z 260.75, A 0, B 90, C 0, E1 0, E2 0, E3 0, E4 0} C_DIS
LIN {X -94.197, Y 25.277, Z 260.75, A 0, B 90, C 0, E1 0, E2 0, E3 0, E4 0} C_DIS
LIN {X -94.5, Y 29.229, Z 260.75, A 0, B 90, C 0, E1 0, E2 0, E3 0, E4 0} C_DIS
LIN {X -95.083, Y 33.151, Z 260.75, A 0, B 90, C 0, E1 0, E2 0, E3 0, E4 0} C_DIS
LIN {X -95.81, Y 37.049, Z 260.75, A 0, B 90, C 0, E1 0, E2 0, E3 0, E4 0} C_DIS
LIN {X -96.596, Y 40.936, Z 260.75, A 0, B 90, C 0, E1 0, E2 0, E3 0, E4 0} C_DIS
LIN {X -97.375, Y 44.824, Z 260.75, A 0, B 90, C 0, E1 0, E2 0, E3 0, E4 0} C_DIS
LIN {X -98.072, Y 48.728, Z 260.75, A 0, B 90, C 0, E1 0, E2 0, E3 0, E4 0} C_DIS
LIN {X -98.602, Y 52.657, Z 260.75, A 0, B 90, C 0, E1 0, E2 0, E3 0, E4 0} C_DIS
LIN {X -98.859, Y 56.613, Z 260.75, A 0, B 90, C 0, E1 0, E2 0, E3 0, E4 0} C_DIS
LIN {X -98.715, Y 60.574, Z 260.75, A 0, B 90, C 0, E1 0, E2 0, E3 0, E4 0} C_DIS
LIN {X -98.023, Y 64.474, Z 260.75, A 0, B 90, C 0, E1 0, E2 0, E3 0, E4 0} C_DIS
LIN {X -96.656, Y 68.19, Z 260.75, A 0, B 90, C 0, E1 0, E2 0, E3 0, E4 0} C_DIS
LIN {X -94.584, Y 71.563, Z 260.75, A 0, B 90, C 0, E1 0, E2 0, E3 0, E4 0} C_DIS
LIN {X -91.91, Y 74.484, Z 260.75, A 0, B 90, C 0, E1 0, E2 0, E3 0, E4 0} C_DIS
LIN {X -88.799, Y 76.938, Z 260.75, A 0, B 90, C 0, E1 0, E2 0, E3 0, E4 0} C_DIS
LIN {X -85.4, Y 78.977, Z 260.75, A 0, B 90, C 0, E1 0, E2 0, E3 0, E4 0} C_DIS
LIN {X -81.818, Y 80.676, Z 260.75, A 0, B 90, C 0, E1 0, E2 0, E3 0, E4 0} C_DIS
LIN {X -78.124, Y 82.116, Z 260.75, A 0, B 90, C 0, E1 0, E2 0, E3 0, E4 0} C_DIS
LIN {X -74.365, Y 83.376, Z 260.75, A 0, B 90, C 0, E1 0, E2 0, E3 0, E4 0} C_DIS
LIN {X -70.577, Y 84.549, Z 260.75, A 0, B 90, C 0, E1 0, E2 0, E3 0, E4 0} C_DIS
LIN {X -66.799, Y 85.756, Z 260.75, A 0, B 90, C 0, E1 0, E2 0, E3 0, E4 0} C_DIS
LIN {X -63.101, Y 87.183, Z 260.75, A 0, B 90, C 0, E1 0, E2 0, E3 0, E4 0} C_DIS
LIN {X -59.635, Y 89.098, Z 260.75, A 0, B 90, C 0, E1 0, E2 0, E3 0, E4 0} C_DIS
LIN {X -56.643, Y 91.689, Z 260.75, A 0, B 90, C 0, E1 0, E2 0, E3 0, E4 0} C_DIS
LIN {X -54.183, Y 94.794, Z 260.75, A 0, B 90, C 0, E1 0, E2 0, E3 0, E4 0} C_DIS
LIN {X -52.048, Y 98.135, Z 260.75, A 0, B 90, C 0, E1 0, E2 0, E3 0, E4 0} C_DIS
LIN {X -50.027, Y 101.547, Z 260.75, A 0, B 90, C 0, E1 0, E2 0, E3 0, E4 0} C_DIS
LIN {X -47.984, Y 104.945, Z 260.75, A 0, B 90, C 0, E1 0, E2 0, E3 0, E4 0} C_DIS
LIN {X -45.829, Y 108.274, Z 260.75, A 0, B 90, C 0, E1 0, E2 0, E3 0, E4 0} C_DIS
LIN {X -43.5, Y 111.483, Z 260.75, A 0, B 90, C 0, E1 0, E2 0, E3 0, E4 0} C_DIS
LIN {X -40.947, Y 114.516, Z 260.75, A 0, B 90, C 0, E1 0, E2 0, E3 0, E4 0} C_DIS
LIN {X -38.128, Y 117.302, Z 260.75, A 0, B 90, C 0, E1 0, E2 0, E3 0, E4 0} C_DIS
LIN {X -35.006, Y 119.742, Z 260.75, A 0, B 90, C 0, E1 0, E2 0, E3 0, E4 0} C_DIS
LIN {X -31.563, Y 121.701, Z 260.75, A 0, B 90, C 0, E1 0, E2 0, E3 0, E4 0} C_DIS
LIN {X -27.827, Y 123.012, Z 260.75, A 0, B 90, C 0, E1 0, E2 0, E3 0, E4 0} C_DIS
LIN {X -23.903, Y 123.527, Z 260.75, A 0, B 90, C 0, E1 0, E2 0, E3 0, E4 0} C_DIS
LIN {X -19.957, Y 123.21, Z 260.75, A 0, B 90, C 0, E1 0, E2 0, E3 0, E4 0} C_DIS
LIN {X -16.137, Y 122.163, Z 260.75, A 0, B 90, C 0, E1 0, E2 0, E3 0, E4 0} C_DIS
LIN {X -12.516, Y 120.553, Z 260.75, A 0, B 90, C 0, E1 0, E2 0, E3 0, E4 0} C_DIS
LIN {X -9.106, Y 118.533, Z 260.75, A 0, B 90, C 0, E1 0, E2 0, E3 0, E4 0} C_DIS
LIN {X -5.892, Y 116.213, Z 260.75, A 0, B 90, C 0, E1 0, E2 0, E3 0, E4 0} C_DIS
LIN {X -2.854, Y 113.668, Z 260.75, A 0, B 90, C 0, E1 0, E2 0, E3 0, E4 0} C_DIS
LIN {X 0, Y 111.06, Z 260.75, A 0, B 90, C 0, E1 0, E2 0, E3 0, E4 0} C_DIS
LIN {X 2.491, Y 108.272, Z 260.75, A 0, B 90, C 0, E1 0, E2 0, E3 0, E4 0} C_DIS
LIN {X 5.284, Y 105.459, Z 260.75, A 0, B 90, C 0, E1 0, E2 0, E3 0, E4 0} C_DIS
LIN {X 8.097, Y 102.664, Z 260.75, A 0, B 90, C 0, E1 0, E2 0, E3 0, E4 0} C_DIS
LIN {X 10.989, Y 99.951, Z 260.75, A 0, B 90, C 0, E1 0, E2 0, E3 0, E4 0} C_DIS
LIN {X 14.079, Y 97.469, Z 260.75, A 0, B 90, C 0, E1 0, E2 0, E3 0, E4 0} C_DIS
LIN {X 17.52, Y 95.512, Z 260.75, A 0, B 90, C 0, E1 0, E2 0, E3 0, E4 0} C_DIS
LIN {X 21.323, Y 94.427, Z 260.75, A 0, B 90, C 0, E1 0, E2 0, E3 0, E4 0} C_DIS
LIN {X 25.277, Y 94.197, Z 260.75, A 0, B 90, C 0, E1 0, E2 0, E3 0, E4 0} C_DIS
LIN {X 29.229, Y 94.5, Z 260.75, A 0, B 90, C 0, E1 0, E2 0, E3 0, E4 0} C_DIS
LIN {X 33.151, Y 95.083, Z 260.75, A 0, B 90, C 0, E1 0, E2 0, E3 0, E4 0} C_DIS
LIN {X 37.049, Y 95.81, Z 260.75, A 0, B 90, C 0, E1 0, E2 0, E3 0, E4 0} C_DIS
LIN {X 40.936, Y 96.596, Z 260.75, A 0, B 90, C 0, E1 0, E2 0, E3 0, E4 0} C_DIS
LIN {X 44.824, Y 97.375, Z 260.75, A 0, B 90, C 0, E1 0, E2 0, E3 0, E4 0} C_DIS
LIN {X 48.728, Y 98.072, Z 260.75, A 0, B 90, C 0, E1 0, E2 0, E3 0, E4 0} C_DIS
LIN {X 52.657, Y 98.602, Z 260.75, A 0, B 90, C 0, E1 0, E2 0, E3 0, E4 0} C_DIS
LIN {X 56.613, Y 98.859, Z 260.75, A 0, B 90, C 0, E1 0, E2 0, E3 0, E4 0} C_DIS
LIN {X 60.574, Y 98.715, Z 260.75, A 0, B 90, C 0, E1 0, E2 0, E3 0, E4 0} C_DIS
LIN {X 64.474, Y 98.023, Z 260.75, A 0, B 90, C 0, E1 0, E2 0, E3 0, E4 0} C_DIS
LIN {X 68.19, Y 96.656, Z 260.75, A 0, B 90, C 0, E1 0, E2 0, E3 0, E4 0} C_DIS
LIN {X 71.563, Y 94.584, Z 260.75, A 0, B 90, C 0, E1 0, E2 0, E3 0, E4 0} C_DIS
LIN {X 74.484, Y 91.91, Z 260.75, A 0, B 90, C 0, E1 0, E2 0, E3 0, E4 0} C_DIS
LIN {X 76.938, Y 88.799, Z 260.75, A 0, B 90, C 0, E1 0, E2 0, E3 0, E4 0} C_DIS
LIN {X 78.977, Y 85.4, Z 260.75, A 0, B 90, C 0, E1 0, E2 0, E3 0, E4 0} C_DIS
LIN {X 80.676, Y 81.818, Z 260.75, A 0, B 90, C 0, E1 0, E2 0, E3 0, E4 0} C_DIS
LIN {X 82.116, Y 78.124, Z 260.75, A 0, B 90, C 0, E1 0, E2 0, E3 0, E4 0} C_DIS
LIN {X 83.376, Y 74.365, Z 260.75, A 0, B 90, C 0, E1 0, E2 0, E3 0, E4 0} C_DIS
LIN {X 84.549, Y 70.577, Z 260.75, A 0, B 90, C 0, E1 0, E2 0, E3 0, E4 0} C_DIS
LIN {X 85.756, Y 66.799, Z 260.75, A 0, B 90, C 0, E1 0, E2 0, E3 0, E4 0} C_DIS
LIN {X 87.183, Y 63.101, Z 260.75, A 0, B 90, C 0, E1 0, E2 0, E3 0, E4 0} C_DIS
LIN {X 89.098, Y 59.635, Z 260.75, A 0, B 90, C 0, E1 0, E2 0, E3 0, E4 0} C_DIS
LIN {X 91.689, Y 56.643, Z 260.75, A 0, B 90, C 0, E1 0, E2 0, E3 0, E4 0} C_DIS
LIN {X 94.794, Y 54.183, Z 260.75, A 0, B 90, C 0, E1 0, E2 0, E3 0, E4 0} C_DIS
LIN {X 98.135, Y 52.048, Z 260.75, A 0, B 90, C 0, E1 0, E2 0, E3 0, E4 0} C_DIS
LIN {X 101.547, Y 50.027, Z 260.75, A 0, B 90, C 0, E1 0, E2 0, E3 0, E4 0} C_DIS
LIN {X 104.945, Y 47.984, Z 260.75, A 0, B 90, C 0, E1 0, E2 0, E3 0, E4 0} C_DIS
LIN {X 108.274, Y 45.829, Z 260.75, A 0, B 90, C 0, E1 0, E2 0, E3 0, E4 0} C_DIS
LIN {X 111.483, Y 43.5, Z 260.75, A 0, B 90, C 0, E1 0, E2 0, E3 0, E4 0} C_DIS
LIN {X 114.516, Y 40.947, Z 260.75, A 0, B 90, C 0, E1 0, E2 0, E3 0, E4 0} C_DIS
LIN {X 117.302, Y 38.128, Z 260.75, A 0, B 90, C 0, E1 0, E2 0, E3 0, E4 0} C_DIS
LIN {X 119.742, Y 35.006, Z 260.75, A 0, B 90, C 0, E1 0, E2 0, E3 0, E4 0} C_DIS
LIN {X 121.701, Y 31.563, Z 260.75, A 0, B 90, C 0, E1 0, E2 0, E3 0, E4 0} C_DIS
LIN {X 123.012, Y 27.827, Z 260.75, A 0, B 90, C 0, E1 0, E2 0, E3 0, E4 0} C_DIS
LIN {X 123.527, Y 23.903, Z 260.75, A 0, B 90, C 0, E1 0, E2 0, E3 0, E4 0} C_DIS
LIN {X 123.21, Y 19.957, Z 260.75, A 0, B 90, C 0, E1 0, E2 0, E3 0, E4 0} C_DIS
LIN {X 122.163, Y 16.137, Z 260.75, A 0, B 90, C 0, E1 0, E2 0, E3 0, E4 0} C_DIS
LIN {X 120.553, Y 12.516, Z 260.75, A 0, B 90, C 0, E1 0, E2 0, E3 0, E4 0} C_DIS
LIN {X 118.533, Y 9.106, Z 260.75, A 0, B 90, C 0, E1 0, E2 0, E3 0, E4 0} C_DIS
LIN {X 116.213, Y 5.892, Z 260.75, A 0, B 90, C 0, E1 0, E2 0, E3 0, E4 0} C_DIS
LIN {X 113.668, Y 2.854, Z 260.75, A 0, B 90, C 0, E1 0, E2 0, E3 0, E4 0} C_DIS
LIN {X 111.06, Y 0, Z 260.75, A 0, B 90, C 0, E1 0, E2 0, E3 0, E4 0} C_DIS
LIN {X 108.272, Y -2.491, Z 260.75, A 0, B 90, C 0, E1 0, E2 0, E3 0, E4 0} C_DIS
LIN {X 105.459, Y -5.284, Z 260.75, A 0, B 90, C 0, E1 0, E2 0, E3 0, E4 0} C_DIS
LIN {X 102.664, Y -8.097, Z 260.75, A 0, B 90, C 0, E1 0, E2 0, E3 0, E4 0} C_DIS
LIN {X 99.951, Y -10.989, Z 260.75, A 0, B 90, C 0, E1 0, E2 0, E3 0, E4 0} C_DIS
LIN {X 97.469, Y -14.079, Z 260.75, A 0, B 90, C 0, E1 0, E2 0, E3 0, E4 0} C_DIS
LIN {X 95.512, Y -17.52, Z 260.75, A 0, B 90, C 0, E1 0, E2 0, E3 0, E4 0} C_DIS
LIN {X 94.427, Y -21.323, Z 260.75, A 0, B 90, C 0, E1 0, E2 0, E3 0, E4 0} C_DIS
LIN {X 94.197, Y -25.277, Z 260.75, A 0, B 90, C 0, E1 0, E2 0, E3 0, E4 0} C_DIS
LIN {X 94.5, Y -29.229, Z 260.75, A 0, B 90, C 0, E1 0, E2 0, E3 0, E4 0} C_DIS
LIN {X 95.083, Y -33.151, Z 260.75, A 0, B 90, C 0, E1 0, E2 0, E3 0, E4 0} C_DIS
LIN {X 95.81, Y -37.049, Z 260.75, A 0, B 90, C 0, E1 0, E2 0, E3 0, E4 0} C_DIS
LIN {X 96.596, Y -40.936, Z 260.75, A 0, B 90, C 0, E1 0, E2 0, E3 0, E4 0} C_DIS
LIN {X 97.375, Y -44.824, Z 260.75, A 0, B 90, C 0, E1 0, E2 0, E3 0, E4 0} C_DIS
LIN {X 98.072, Y -48.728, Z 260.75, A 0, B 90, C 0, E1 0, E2 0, E3 0, E4 0} C_DIS
LIN {X 98.602, Y -52.657, Z 260.75, A 0, B 90, C 0, E1 0, E2 0, E3 0, E4 0} C_DIS
LIN {X 98.859, Y -56.613, Z 260.75, A 0, B 90, C 0, E1 0, E2 0, E3 0, E4 0} C_DIS
LIN {X 98.715, Y -60.574, Z 260.75, A 0, B 90, C 0, E1 0, E2 0, E3 0, E4 0} C_DIS
LIN {X 98.023, Y -64.474, Z 260.75, A 0, B 90, C 0, E1 0, E2 0, E3 0, E4 0} C_DIS
LIN {X 96.656, Y -68.19, Z 260.75, A 0, B 90, C 0, E1 0, E2 0, E3 0, E4 0} C_DIS
LIN {X 94.584, Y -71.563, Z 260.75, A 0, B 90, C 0, E1 0, E2 0, E3 0, E4 0} C_DIS
LIN {X 91.91, Y -74.484, Z 260.75, A 0, B 90, C 0, E1 0, E2 0, E3 0, E4 0} C_DIS
LIN {X 88.799, Y -76.938, Z 260.75, A 0, B 90, C 0, E1 0, E2 0, E3 0, E4 0} C_DIS
LIN {X 85.4, Y -78.977, Z 260.75, A 0, B 90, C 0, E1 0, E2 0, E3 0, E4 0} C_DIS
LIN {X 81.818, Y -80.676, Z 260.75, A 0, B 90, C 0, E1 0, E2 0, E3 0, E4 0} C_DIS
LIN {X 78.124, Y -82.116, Z 260.75, A 0, B 90, C 0, E1 0, E2 0, E3 0, E4 0} C_DIS
LIN {X 74.365, Y -83.376, Z 260.75, A 0, B 90, C 0, E1 0, E2 0, E3 0, E4 0} C_DIS
LIN {X 70.577, Y -84.549, Z 260.75, A 0, B 90, C 0, E1 0, E2 0, E3 0, E4 0} C_DIS
LIN {X 66.799, Y -85.756, Z 260.75, A 0, B 90, C 0, E1 0, E2 0, E3 0, E4 0} C_DIS
LIN {X 63.101, Y -87.183, Z 260.75, A 0, B 90, C 0, E1 0, E2 0, E3 0, E4 0} C_DIS
LIN {X 59.635, Y -89.098, Z 260.75, A 0, B 90, C 0, E1 0, E2 0, E3 0, E4 0} C_DIS
LIN {X 56.643, Y -91.689, Z 260.75, A 0, B 90, C 0, E1 0, E2 0, E3 0, E4 0} C_DIS
LIN {X 54.183, Y -94.794, Z 260.75, A 0, B 90, C 0, E1 0, E2 0, E3 0, E4 0} C_DIS
LIN {X 52.048, Y -98.135, Z 260.75, A 0, B 90, C 0, E1 0, E2 0, E3 0, E4 0} C_DIS
LIN {X 50.027, Y -101.547, Z 260.75, A 0, B 90, C 0, E1 0, E2 0, E3 0, E4 0} C_DIS
LIN {X 47.984, Y -104.945, Z 260.75, A 0, B 90, C 0, E1 0, E2 0, E3 0, E4 0} C_DIS
LIN {X 45.829, Y -108.274, Z 260.75, A 0, B 90, C 0, E1 0, E2 0, E3 0, E4 0} C_DIS
LIN {X 43.5, Y -111.483, Z 260.75, A 0, B 90, C 0, E1 0, E2 0, E3 0, E4 0} C_DIS
LIN {X 40.947, Y -114.516, Z 260.75, A 0, B 90, C 0, E1 0, E2 0, E3 0, E4 0} C_DIS
LIN {X 38.128, Y -117.302, Z 260.75, A 0, B 90, C 0, E1 0, E2 0, E3 0, E4 0} C_DIS
LIN {X 35.006, Y -119.742, Z 260.75, A 0, B 90, C 0, E1 0, E2 0, E3 0, E4 0} C_DIS
LIN {X 31.563, Y -121.701, Z 260.75, A 0, B 90, C 0, E1 0, E2 0, E3 0, E4 0} C_DIS
LIN {X 27.827, Y -123.012, Z 260.75, A 0, B 90, C 0, E1 0, E2 0, E3 0, E4 0} C_DIS
LIN {X 23.903, Y -123.527, Z 260.75, A 0, B 90, C 0, E1 0, E2 0, E3 0, E4 0} C_DIS
LIN {X 19.957, Y -123.21, Z 260.75, A 0, B 90, C 0, E1 0, E2 0, E3 0, E4 0} C_DIS
LIN {X 16.137, Y -122.163, Z 260.75, A 0, B 90, C 0, E1 0, E2 0, E3 0, E4 0} C_DIS
LIN {X 12.516, Y -120.553, Z 260.75, A 0, B 90, C 0, E1 0, E2 0, E3 0, E4 0} C_DIS
LIN {X 9.106, Y -118.533, Z 260.75, A 0, B 90, C 0, E1 0, E2 0, E3 0, E4 0} C_DIS
LIN {X 5.892, Y -116.213, Z 260.75, A 0, B 90, C 0, E1 0, E2 0, E3 0, E4 0} C_DIS
LIN {X 2.854, Y -113.668, Z 260.75, A 0, B 90, C 0, E1 0, E2 0, E3 0, E4 0} C_DIS
LIN {X 0, Y -111.06, Z 260.75, A 0, B 90, C 0, E1 0, E2 0, E3 0, E4 0} C_DIS
LIN {X -2.491, Y -108.272, Z 260.75, A 0, B 90, C 0, E1 0, E2 0, E3 0, E4 0} C_DIS
LIN {X -5.284, Y -105.459, Z 260.75, A 0, B 90, C 0, E1 0, E2 0, E3 0, E4 0} C_DIS
LIN {X -8.097, Y -102.664, Z 260.75, A 0, B 90, C 0, E1 0, E2 0, E3 0, E4 0} C_DIS
LIN {X -10.989, Y -99.951, Z 260.75, A 0, B 90, C 0, E1 0, E2 0, E3 0, E4 0} C_DIS
LIN {X -14.079, Y -97.469, Z 260.75, A 0, B 90, C 0, E1 0, E2 0, E3 0, E4 0} C_DIS
LIN {X -17.52, Y -95.512, Z 260.75, A 0, B 90, C 0, E1 0, E2 0, E3 0, E4 0} C_DIS
LIN {X -21.323, Y -94.427, Z 260.75, A 0, B 90, C 0, E1 0, E2 0, E3 0, E4 0} C_DIS
LIN {X -25.277, Y -94.197, Z 260.75, A 0, B 90, C 0, E1 0, E2 0, E3 0, E4 0} C_DIS
LIN {X -29.229, Y -94.5, Z 260.75, A 0, B 90, C 0, E1 0, E2 0, E3 0, E4 0} C_DIS
LIN {X -33.151, Y -95.083, Z 260.75, A 0, B 90, C 0, E1 0, E2 0, E3 0, E4 0} C_DIS
LIN {X -37.049, Y -95.81, Z 260.75, A 0, B 90, C 0, E1 0, E2 0, E3 0, E4 0} C_DIS
LIN {X -40.936, Y -96.596, Z 260.75, A 0, B 90, C 0, E1 0, E2 0, E3 0, E4 0} C_DIS
LIN {X -44.824, Y -97.375, Z 260.75, A 0, B 90, C 0, E1 0, E2 0, E3 0, E4 0} C_DIS
LIN {X -48.728, Y -98.072, Z 260.75, A 0, B 90, C 0, E1 0, E2 0, E3 0, E4 0} C_DIS
LIN {X -52.657, Y -98.602, Z 260.75, A 0, B 90, C 0, E1 0, E2 0, E3 0, E4 0} C_DIS
LIN {X -56.613, Y -98.859, Z 260.75, A 0, B 90, C 0, E1 0, E2 0, E3 0, E4 0} C_DIS
LIN {X -60.574, Y -98.715, Z 260.75, A 0, B 90, C 0, E1 0, E2 0, E3 0, E4 0} C_DIS
LIN {X -64.474, Y -98.023, Z 260.75, A 0, B 90, C 0, E1 0, E2 0, E3 0, E4 0} C_DIS
LIN {X -68.19, Y -96.656, Z 260.75, A 0, B 90, C 0, E1 0, E2 0, E3 0, E4 0} C_DIS
LIN {X -71.563, Y -94.584, Z 260.75, A 0, B 90, C 0, E1 0, E2 0, E3 0, E4 0} C_DIS
LIN {X -74.484, Y -91.91, Z 260.75, A 0, B 90, C 0, E1 0, E2 0, E3 0, E4 0} C_DIS
LIN {X -76.938, Y -88.799, Z 260.75, A 0, B 90, C 0, E1 0, E2 0, E3 0, E4 0} C_DIS
LIN {X -78.977, Y -85.4, Z 260.75, A 0, B 90, C 0, E1 0, E2 0, E3 0, E4 0} C_DIS
LIN {X -80.676, Y -81.818, Z 260.75, A 0, B 90, C 0, E1 0, E2 0, E3 0, E4 0} C_DIS
LIN {X -82.116, Y -78.124, Z 260.75, A 0, B 90, C 0, E1 0, E2 0, E3 0, E4 0} C_DIS
LIN {X -83.376, Y -74.365, Z 260.75, A 0, B 90, C 0, E1 0, E2 0, E3 0, E4 0} C_DIS
LIN {X -84.549, Y -70.577, Z 260.75, A 0, B 90, C 0, E1 0, E2 0, E3 0, E4 0} C_DIS
LIN {X -85.756, Y -66.799, Z 260.75, A 0, B 90, C 0, E1 0, E2 0, E3 0, E4 0} C_DIS
LIN {X -87.183, Y -63.101, Z 260.75, A 0, B 90, C 0, E1 0, E2 0, E3 0, E4 0} C_DIS
LIN {X -89.098, Y -59.635, Z 260.75, A 0, B 90, C 0, E1 0, E2 0, E3 0, E4 0} C_DIS
LIN {X -91.689, Y -56.643, Z 260.75, A 0, B 90, C 0, E1 0, E2 0, E3 0, E4 0} C_DIS
LIN {X -94.794, Y -54.183, Z 260.75, A 0, B 90, C 0, E1 0, E2 0, E3 0, E4 0} C_DIS
LIN {X -98.135, Y -52.048, Z 260.75, A 0, B 90, C 0, E1 0, E2 0, E3 0, E4 0} C_DIS
LIN {X -101.547, Y -50.027, Z 260.75, A 0, B 90, C 0, E1 0, E2 0, E3 0, E4 0} C_DIS
LIN {X -104.945, Y -47.984, Z 260.75, A 0, B 90, C 0, E1 0, E2 0, E3 0, E4 0} C_DIS
LIN {X -108.274, Y -45.829, Z 260.75, A 0, B 90, C 0, E1 0, E2 0, E3 0, E4 0} C_DIS
LIN {X -111.483, Y -43.5, Z 260.75, A 0, B 90, C 0, E1 0, E2 0, E3 0, E4 0} C_DIS
LIN {X -114.516, Y -40.947, Z 260.75, A 0, B 90, C 0, E1 0, E2 0, E3 0, E4 0} C_DIS
LIN {X -117.302, Y -38.128, Z 260.75, A 0, B 90, C 0, E1 0, E2 0, E3 0, E4 0} C_DIS
LIN {X -119.742, Y -35.006, Z 260.75, A 0, B 90, C 0, E1 0, E2 0, E3 0, E4 0} C_DIS
LIN {X -121.701, Y -31.563, Z 260.75, A 0, B 90, C 0, E1 0, E2 0, E3 0, E4 0} C_DIS
LIN {X -123.012, Y -27.827, Z 260.75, A 0, B 90, C 0, E1 0, E2 0, E3 0, E4 0} C_DIS
LIN {X -123.527, Y -23.903, Z 260.75, A 0, B 90, C 0, E1 0, E2 0, E3 0, E4 0} C_DIS
LIN {X -123.21, Y -19.957, Z 260.75, A 0, B 90, C 0, E1 0, E2 0, E3 0, E4 0} C_DIS
LIN {X -122.163, Y -16.137, Z 260.75, A 0, B 90, C 0, E1 0, E2 0, E3 0, E4 0} C_DIS
LIN {X -120.553, Y -12.516, Z 260.75, A 0, B 90, C 0, E1 0, E2 0, E3 0, E4 0} C_DIS
LIN {X -118.533, Y -9.106, Z 260.75, A 0, B 90, C 0, E1 0, E2 0, E3 0, E4 0} C_DIS
LIN {X -116.213, Y -5.892, Z 260.75, A 0, B 90, C 0, E1 0, E2 0, E3 0, E4 0} C_DIS
LIN {X -113.668, Y -2.854, Z 260.75, A 0, B 90, C 0, E1 0, E2 0, E3 0, E4 0} C_DIS
LIN {X -111.873, Y 0, Z 263.25, A 0, B 90, C 0, E1 0, E2 0, E3 0, E4 0} C_DIS
LIN {X -109.049, Y 2.52, Z 263.25, A 0, B 90, C 0, E1 0, E2 0, E3 0, E4 0} C_DIS
LIN {X -106.199, Y 5.337, Z 263.25, A 0, B 90, C 0, E1 0, E2 0, E3 0, E4 0} C_DIS
LIN {X -103.369, Y 8.176, Z 263.25, A 0, B 90, C 0, E1 0, E2 0, E3 0, E4 0} C_DIS
LIN {X -100.625, Y 11.097, Z 263.25, A 0, B 90, C 0, E1 0, E2 0, E3 0, E4 0} C_DIS
LIN {X -98.125, Y 14.229, Z 263.25, A 0, B 90, C 0, E1 0, E2 0, E3 0, E4 0} C_DIS
LIN {X -96.177, Y 17.724, Z 263.25, A 0, B 90, C 0, E1 0, E2 0, E3 0, E4 0} C_DIS
LIN {X -95.14, Y 21.584, Z 263.25, A 0, B 90, C 0, E1 0, E2 0, E3 0, E4 0} C_DIS
LIN {X -94.985, Y 25.585, Z 263.25, A 0, B 90, C 0, E1 0, E2 0, E3 0, E4 0} C_DIS
LIN {X -95.37, Y 29.573, Z 263.25, A 0, B 90, C 0, E1 0, E2 0, E3 0, E4 0} C_DIS
LIN {X -96.035, Y 33.526, Z 263.25, A 0, B 90, C 0, E1 0, E2 0, E3 0, E4 0} C_DIS
LIN {X -96.835, Y 37.454, Z 263.25, A 0, B 90, C 0, E1 0, E2 0, E3 0, E4 0} C_DIS
LIN {X -97.687, Y 41.372, Z 263.25, A 0, B 90, C 0, E1 0, E2 0, E3 0, E4 0} C_DIS
LIN {X -98.518, Y 45.293, Z 263.25, A 0, B 90, C 0, E1 0, E2 0, E3 0, E4 0} C_DIS
LIN {X -99.257, Y 49.233, Z 263.25, A 0, B 90, C 0, E1 0, E2 0, E3 0, E4 0} C_DIS
LIN {X -99.813, Y 53.203, Z 263.25, A 0, B 90, C 0, E1 0, E2 0, E3 0, E4 0} C_DIS
LIN {X -100.081, Y 57.201, Z 263.25, A 0, B 90, C 0, E1 0, E2 0, E3 0, E4 0} C_DIS
LIN {X -99.928, Y 61.204, Z 263.25, A 0, B 90, C 0, E1 0, E2 0, E3 0, E4 0} C_DIS
LIN {X -99.201, Y 65.142, Z 263.25, A 0, B 90, C 0, E1 0, E2 0, E3 0, E4 0} C_DIS
LIN {X -97.773, Y 68.881, Z 263.25, A 0, B 90, C 0, E1 0, E2 0, E3 0, E4 0} C_DIS
LIN {X -95.62, Y 72.254, Z 263.25, A 0, B 90, C 0, E1 0, E2 0, E3 0, E4 0} C_DIS
LIN {X -92.854, Y 75.148, Z 263.25, A 0, B 90, C 0, E1 0, E2 0, E3 0, E4 0} C_DIS
LIN {X -89.651, Y 77.553, Z 263.25, A 0, B 90, C 0, E1 0, E2 0, E3 0, E4 0} C_DIS
LIN {X -86.165, Y 79.527, Z 263.25, A 0, B 90, C 0, E1 0, E2 0, E3 0, E4 0} C_DIS
LIN {X -82.501, Y 81.152, Z 263.25, A 0, B 90, C 0, E1 0, E2 0, E3 0, E4 0} C_DIS
LIN {X -78.731, Y 82.512, Z 263.25, A 0, B 90, C 0, E1 0, E2 0, E3 0, E4 0} C_DIS
LIN {X -74.9, Y 83.692, Z 263.25, A 0, B 90, C 0, E1 0, E2 0, E3 0, E4 0} C_DIS
LIN {X -71.043, Y 84.787, Z 263.25, A 0, B 90, C 0, E1 0, E2 0, E3 0, E4 0} C_DIS
LIN {X -67.199, Y 85.921, Z 263.25, A 0, B 90, C 0, E1 0, E2 0, E3 0, E4 0} C_DIS
LIN {X -63.432, Y 87.287, Z 263.25, A 0, B 90, C 0, E1 0, E2 0, E3 0, E4 0} C_DIS
LIN {X -59.897, Y 89.165, Z 263.25, A 0, B 90, C 0, E1 0, E2 0, E3 0, E4 0} C_DIS
LIN {X -56.847, Y 91.754, Z 263.25, A 0, B 90, C 0, E1 0, E2 0, E3 0, E4 0} C_DIS
LIN {X -54.356, Y 94.889, Z 263.25, A 0, B 90, C 0, E1 0, E2 0, E3 0, E4 0} C_DIS
LIN {X -52.215, Y 98.278, Z 263.25, A 0, B 90, C 0, E1 0, E2 0, E3 0, E4 0} C_DIS
LIN {X -50.205, Y 101.746, Z 263.25, A 0, B 90, C 0, E1 0, E2 0, E3 0, E4 0} C_DIS
LIN {X -48.182, Y 105.207, Z 263.25, A 0, B 90, C 0, E1 0, E2 0, E3 0, E4 0} C_DIS
LIN {X -46.052, Y 108.603, Z 263.25, A 0, B 90, C 0, E1 0, E2 0, E3 0, E4 0} C_DIS
LIN {X -43.751, Y 111.885, Z 263.25, A 0, B 90, C 0, E1 0, E2 0, E3 0, E4 0} C_DIS
LIN {X -41.226, Y 114.997, Z 263.25, A 0, B 90, C 0, E1 0, E2 0, E3 0, E4 0} C_DIS
LIN {X -38.429, Y 117.867, Z 263.25, A 0, B 90, C 0, E1 0, E2 0, E3 0, E4 0} C_DIS
LIN {X -35.322, Y 120.394, Z 263.25, A 0, B 90, C 0, E1 0, E2 0, E3 0, E4 0} C_DIS
LIN {X -31.88, Y 122.441, Z 263.25, A 0, B 90, C 0, E1 0, E2 0, E3 0, E4 0} C_DIS
LIN {X -28.128, Y 123.833, Z 263.25, A 0, B 90, C 0, E1 0, E2 0, E3 0, E4 0} C_DIS
LIN {X -24.169, Y 124.411, Z 263.25, A 0, B 90, C 0, E1 0, E2 0, E3 0, E4 0} C_DIS
LIN {X -20.177, Y 124.132, Z 263.25, A 0, B 90, C 0, E1 0, E2 0, E3 0, E4 0} C_DIS
LIN {X -16.309, Y 123.098, Z 263.25, A 0, B 90, C 0, E1 0, E2 0, E3 0, E4 0} C_DIS
LIN {X -12.643, Y 121.482, Z 263.25, A 0, B 90, C 0, E1 0, E2 0, E3 0, E4 0} C_DIS
LIN {X -9.195, Y 119.442, Z 263.25, A 0, B 90, C 0, E1 0, E2 0, E3 0, E4 0} C_DIS
LIN {X -5.947, Y 117.095, Z 263.25, A 0, B 90, C 0, E1 0, E2 0, E3 0, E4 0} C_DIS
LIN {X -2.879, Y 114.518, Z 263.25, A 0, B 90, C 0, E1 0, E2 0, E3 0, E4 0} C_DIS
LIN {X 0, Y 111.873, Z 263.25, A 0, B 90, C 0, E1 0, E2 0, E3 0, E4 0} C_DIS
LIN {X 2.52, Y 109.049, Z 263.25, A 0, B 90, C 0, E1 0, E2 0, E3 0, E4 0} C_DIS
LIN {X 5.337, Y 106.199, Z 263.25, A 0, B 90, C 0, E1 0, E2 0, E3 0, E4 0} C_DIS
LIN {X 8.176, Y 103.369, Z 263.25, A 0, B 90, C 0, E1 0, E2 0, E3 0, E4 0} C_DIS
LIN {X 11.097, Y 100.625, Z 263.25, A 0, B 90, C 0, E1 0, E2 0, E3 0, E4 0} C_DIS
LIN {X 14.229, Y 98.125, Z 263.25, A 0, B 90, C 0, E1 0, E2 0, E3 0, E4 0} C_DIS
LIN {X 17.724, Y 96.177, Z 263.25, A 0, B 90, C 0, E1 0, E2 0, E3 0, E4 0} C_DIS
LIN {X 21.584, Y 95.14, Z 263.25, A 0, B 90, C 0, E1 0, E2 0, E3 0, E4 0} C_DIS
LIN {X 25.585, Y 94.985, Z 263.25, A 0, B 90, C 0, E1 0, E2 0, E3 0, E4 0} C_DIS
LIN {X 29.573, Y 95.37, Z 263.25, A 0, B 90, C 0, E1 0, E2 0, E3 0, E4 0} C_DIS
LIN {X 33.526, Y 96.035, Z 263.25, A 0, B 90, C 0, E1 0, E2 0, E3 0, E4 0} C_DIS
LIN {X 37.454, Y 96.835, Z 263.25, A 0, B 90, C 0, E1 0, E2 0, E3 0, E4 0} C_DIS
LIN {X 41.372, Y 97.687, Z 263.25, A 0, B 90, C 0, E1 0, E2 0, E3 0, E4 0} C_DIS
LIN {X 45.293, Y 98.518, Z 263.25, A 0, B 90, C 0, E1 0, E2 0, E3 0, E4 0} C_DIS
LIN {X 49.233, Y 99.257, Z 263.25, A 0, B 90, C 0, E1 0, E2 0, E3 0, E4 0} C_DIS
LIN {X 53.203, Y 99.813, Z 263.25, A 0, B 90, C 0, E1 0, E2 0, E3 0, E4 0} C_DIS
LIN {X 57.201, Y 100.081, Z 263.25, A 0, B 90, C 0, E1 0, E2 0, E3 0, E4 0} C_DIS
LIN {X 61.204, Y 99.928, Z 263.25, A 0, B 90, C 0, E1 0, E2 0, E3 0, E4 0} C_DIS
LIN {X 65.142, Y 99.201, Z 263.25, A 0, B 90, C 0, E1 0, E2 0, E3 0, E4 0} C_DIS
LIN {X 68.881, Y 97.773, Z 263.25, A 0, B 90, C 0, E1 0, E2 0, E3 0, E4 0} C_DIS
LIN {X 72.254, Y 95.62, Z 263.25, A 0, B 90, C 0, E1 0, E2 0, E3 0, E4 0} C_DIS
LIN {X 75.148, Y 92.854, Z 263.25, A 0, B 90, C 0, E1 0, E2 0, E3 0, E4 0} C_DIS
LIN {X 77.553, Y 89.651, Z 263.25, A 0, B 90, C 0, E1 0, E2 0, E3 0, E4 0} C_DIS
LIN {X 79.527, Y 86.165, Z 263.25, A 0, B 90, C 0, E1 0, E2 0, E3 0, E4 0} C_DIS
LIN {X 81.152, Y 82.501, Z 263.25, A 0, B 90, C 0, E1 0, E2 0, E3 0, E4 0} C_DIS
LIN {X 82.512, Y 78.731, Z 263.25, A 0, B 90, C 0, E1 0, E2 0, E3 0, E4 0} C_DIS
LIN {X 83.692, Y 74.9, Z 263.25, A 0, B 90, C 0, E1 0, E2 0, E3 0, E4 0} C_DIS
LIN {X 84.787, Y 71.043, Z 263.25, A 0, B 90, C 0, E1 0, E2 0, E3 0, E4 0} C_DIS
LIN {X 85.921, Y 67.199, Z 263.25, A 0, B 90, C 0, E1 0, E2 0, E3 0, E4 0} C_DIS
LIN {X 87.287, Y 63.432, Z 263.25, A 0, B 90, C 0, E1 0, E2 0, E3 0, E4 0} C_DIS
LIN {X 89.165, Y 59.897, Z 263.25, A 0, B 90, C 0, E1 0, E2 0, E3 0, E4 0} C_DIS
LIN {X 91.754, Y 56.847, Z 263.25, A 0, B 90, C 0, E1 0, E2 0, E3 0, E4 0} C_DIS
LIN {X 94.889, Y 54.356, Z 263.25, A 0, B 90, C 0, E1 0, E2 0, E3 0, E4 0} C_DIS
LIN {X 98.278, Y 52.215, Z 263.25, A 0, B 90, C 0, E1 0, E2 0, E3 0, E4 0} C_DIS
LIN {X 101.746, Y 50.205, Z 263.25, A 0, B 90, C 0, E1 0, E2 0, E3 0, E4 0} C_DIS
LIN {X 105.207, Y 48.182, Z 263.25, A 0, B 90, C 0, E1 0, E2 0, E3 0, E4 0} C_DIS
LIN {X 108.603, Y 46.052, Z 263.25, A 0, B 90, C 0, E1 0, E2 0, E3 0, E4 0} C_DIS
LIN {X 111.885, Y 43.751, Z 263.25, A 0, B 90, C 0, E1 0, E2 0, E3 0, E4 0} C_DIS
LIN {X 114.997, Y 41.226, Z 263.25, A 0, B 90, C 0, E1 0, E2 0, E3 0, E4 0} C_DIS
LIN {X 117.867, Y 38.429, Z 263.25, A 0, B 90, C 0, E1 0, E2 0, E3 0, E4 0} C_DIS
LIN {X 120.394, Y 35.322, Z 263.25, A 0, B 90, C 0, E1 0, E2 0, E3 0, E4 0} C_DIS
LIN {X 122.441, Y 31.88, Z 263.25, A 0, B 90, C 0, E1 0, E2 0, E3 0, E4 0} C_DIS
LIN {X 123.833, Y 28.128, Z 263.25, A 0, B 90, C 0, E1 0, E2 0, E3 0, E4 0} C_DIS
LIN {X 124.411, Y 24.169, Z 263.25, A 0, B 90, C 0, E1 0, E2 0, E3 0, E4 0} C_DIS
LIN {X 124.132, Y 20.177, Z 263.25, A 0, B 90, C 0, E1 0, E2 0, E3 0, E4 0} C_DIS
LIN {X 123.098, Y 16.309, Z 263.25, A 0, B 90, C 0, E1 0, E2 0, E3 0, E4 0} C_DIS
LIN {X 121.482, Y 12.643, Z 263.25, A 0, B 90, C 0, E1 0, E2 0, E3 0, E4 0} C_DIS
LIN {X 119.442, Y 9.195, Z 263.25, A 0, B 90, C 0, E1 0, E2 0, E3 0, E4 0} C_DIS
LIN {X 117.095, Y 5.947, Z 263.25, A 0, B 90, C 0, E1 0, E2 0, E3 0, E4 0} C_DIS
LIN {X 114.518, Y 2.879, Z 263.25, A 0, B 90, C 0, E1 0, E2 0, E3 0, E4 0} C_DIS
LIN {X 111.873, Y 0, Z 263.25, A 0, B 90, C 0, E1 0, E2 0, E3 0, E4 0} C_DIS
LIN {X 109.049, Y -2.52, Z 263.25, A 0, B 90, C 0, E1 0, E2 0, E3 0, E4 0} C_DIS
LIN {X 106.199, Y -5.337, Z 263.25, A 0, B 90, C 0, E1 0, E2 0, E3 0, E4 0} C_DIS
LIN {X 103.369, Y -8.176, Z 263.25, A 0, B 90, C 0, E1 0, E2 0, E3 0, E4 0} C_DIS
LIN {X 100.625, Y -11.097, Z 263.25, A 0, B 90, C 0, E1 0, E2 0, E3 0, E4 0} C_DIS
LIN {X 98.125, Y -14.229, Z 263.25, A 0, B 90, C 0, E1 0, E2 0, E3 0, E4 0} C_DIS
LIN {X 96.177, Y -17.724, Z 263.25, A 0, B 90, C 0, E1 0, E2 0, E3 0, E4 0} C_DIS
LIN {X 95.14, Y -21.584, Z 263.25, A 0, B 90, C 0, E1 0, E2 0, E3 0, E4 0} C_DIS
LIN {X 94.985, Y -25.585, Z 263.25, A 0, B 90, C 0, E1 0, E2 0, E3 0, E4 0} C_DIS
LIN {X 95.37, Y -29.573, Z 263.25, A 0, B 90, C 0, E1 0, E2 0, E3 0, E4 0} C_DIS
LIN {X 96.035, Y -33.526, Z 263.25, A 0, B 90, C 0, E1 0, E2 0, E3 0, E4 0} C_DIS
LIN {X 96.835, Y -37.454, Z 263.25, A 0, B 90, C 0, E1 0, E2 0, E3 0, E4 0} C_DIS
LIN {X 97.687, Y -41.372, Z 263.25, A 0, B 90, C 0, E1 0, E2 0, E3 0, E4 0} C_DIS
LIN {X 98.518, Y -45.293, Z 263.25, A 0, B 90, C 0, E1 0, E2 0, E3 0, E4 0} C_DIS
LIN {X 99.257, Y -49.233, Z 263.25, A 0, B 90, C 0, E1 0, E2 0, E3 0, E4 0} C_DIS
LIN {X 99.813, Y -53.203, Z 263.25, A 0, B 90, C 0, E1 0, E2 0, E3 0, E4 0} C_DIS
LIN {X 100.081, Y -57.201, Z 263.25, A 0, B 90, C 0, E1 0, E2 0, E3 0, E4 0} C_DIS
LIN {X 99.928, Y -61.204, Z 263.25, A 0, B 90, C 0, E1 0, E2 0, E3 0, E4 0} C_DIS
LIN {X 99.201, Y -65.142, Z 263.25, A 0, B 90, C 0, E1 0, E2 0, E3 0, E4 0} C_DIS
LIN {X 97.773, Y -68.881, Z 263.25, A 0, B 90, C 0, E1 0, E2 0, E3 0, E4 0} C_DIS
LIN {X 95.62, Y -72.254, Z 263.25, A 0, B 90, C 0, E1 0, E2 0, E3 0, E4 0} C_DIS
LIN {X 92.854, Y -75.148, Z 263.25, A 0, B 90, C 0, E1 0, E2 0, E3 0, E4 0} C_DIS
LIN {X 89.651, Y -77.553, Z 263.25, A 0, B 90, C 0, E1 0, E2 0, E3 0, E4 0} C_DIS
LIN {X 86.165, Y -79.527, Z 263.25, A 0, B 90, C 0, E1 0, E2 0, E3 0, E4 0} C_DIS
LIN {X 82.501, Y -81.152, Z 263.25, A 0, B 90, C 0, E1 0, E2 0, E3 0, E4 0} C_DIS
LIN {X 78.731, Y -82.512, Z 263.25, A 0, B 90, C 0, E1 0, E2 0, E3 0, E4 0} C_DIS
LIN {X 74.9, Y -83.692, Z 263.25, A 0, B 90, C 0, E1 0, E2 0, E3 0, E4 0} C_DIS
LIN {X 71.043, Y -84.787, Z 263.25, A 0, B 90, C 0, E1 0, E2 0, E3 0, E4 0} C_DIS
LIN {X 67.199, Y -85.921, Z 263.25, A 0, B 90, C 0, E1 0, E2 0, E3 0, E4 0} C_DIS
LIN {X 63.432, Y -87.287, Z 263.25, A 0, B 90, C 0, E1 0, E2 0, E3 0, E4 0} C_DIS
LIN {X 59.897, Y -89.165, Z 263.25, A 0, B 90, C 0, E1 0, E2 0, E3 0, E4 0} C_DIS
LIN {X 56.847, Y -91.754, Z 263.25, A 0, B 90, C 0, E1 0, E2 0, E3 0, E4 0} C_DIS
LIN {X 54.356, Y -94.889, Z 263.25, A 0, B 90, C 0, E1 0, E2 0, E3 0, E4 0} C_DIS
LIN {X 52.215, Y -98.278, Z 263.25, A 0, B 90, C 0, E1 0, E2 0, E3 0, E4 0} C_DIS
LIN {X 50.205, Y -101.746, Z 263.25, A 0, B 90, C 0, E1 0, E2 0, E3 0, E4 0} C_DIS
LIN {X 48.182, Y -105.207, Z 263.25, A 0, B 90, C 0, E1 0, E2 0, E3 0, E4 0} C_DIS
LIN {X 46.052, Y -108.603, Z 263.25, A 0, B 90, C 0, E1 0, E2 0, E3 0, E4 0} C_DIS
LIN {X 43.751, Y -111.885, Z 263.25, A 0, B 90, C 0, E1 0, E2 0, E3 0, E4 0} C_DIS
LIN {X 41.226, Y -114.997, Z 263.25, A 0, B 90, C 0, E1 0, E2 0, E3 0, E4 0} C_DIS
LIN {X 38.429, Y -117.867, Z 263.25, A 0, B 90, C 0, E1 0, E2 0, E3 0, E4 0} C_DIS
LIN {X 35.322, Y -120.394, Z 263.25, A 0, B 90, C 0, E1 0, E2 0, E3 0, E4 0} C_DIS
LIN {X 31.88, Y -122.441, Z 263.25, A 0, B 90, C 0, E1 0, E2 0, E3 0, E4 0} C_DIS
LIN {X 28.128, Y -123.833, Z 263.25, A 0, B 90, C 0, E1 0, E2 0, E3 0, E4 0} C_DIS
LIN {X 24.169, Y -124.411, Z 263.25, A 0, B 90, C 0, E1 0, E2 0, E3 0, E4 0} C_DIS
LIN {X 20.177, Y -124.132, Z 263.25, A 0, B 90, C 0, E1 0, E2 0, E3 0, E4 0} C_DIS
LIN {X 16.309, Y -123.098, Z 263.25, A 0, B 90, C 0, E1 0, E2 0, E3 0, E4 0} C_DIS
LIN {X 12.643, Y -121.482, Z 263.25, A 0, B 90, C 0, E1 0, E2 0, E3 0, E4 0} C_DIS
LIN {X 9.195, Y -119.442, Z 263.25, A 0, B 90, C 0, E1 0, E2 0, E3 0, E4 0} C_DIS
LIN {X 5.947, Y -117.095, Z 263.25, A 0, B 90, C 0, E1 0, E2 0, E3 0, E4 0} C_DIS
LIN {X 2.879, Y -114.518, Z 263.25, A 0, B 90, C 0, E1 0, E2 0, E3 0, E4 0} C_DIS
LIN {X 0, Y -111.873, Z 263.25, A 0, B 90, C 0, E1 0, E2 0, E3 0, E4 0} C_DIS
LIN {X -2.52, Y -109.049, Z 263.25, A 0, B 90, C 0, E1 0, E2 0, E3 0, E4 0} C_DIS
LIN {X -5.337, Y -106.199, Z 263.25, A 0, B 90, C 0, E1 0, E2 0, E3 0, E4 0} C_DIS
LIN {X -8.176, Y -103.369, Z 263.25, A 0, B 90, C 0, E1 0, E2 0, E3 0, E4 0} C_DIS
LIN {X -11.097, Y -100.625, Z 263.25, A 0, B 90, C 0, E1 0, E2 0, E3 0, E4 0} C_DIS
LIN {X -14.229, Y -98.125, Z 263.25, A 0, B 90, C 0, E1 0, E2 0, E3 0, E4 0} C_DIS
LIN {X -17.724, Y -96.177, Z 263.25, A 0, B 90, C 0, E1 0, E2 0, E3 0, E4 0} C_DIS
LIN {X -21.584, Y -95.14, Z 263.25, A 0, B 90, C 0, E1 0, E2 0, E3 0, E4 0} C_DIS
LIN {X -25.585, Y -94.985, Z 263.25, A 0, B 90, C 0, E1 0, E2 0, E3 0, E4 0} C_DIS
LIN {X -29.573, Y -95.37, Z 263.25, A 0, B 90, C 0, E1 0, E2 0, E3 0, E4 0} C_DIS
LIN {X -33.526, Y -96.035, Z 263.25, A 0, B 90, C 0, E1 0, E2 0, E3 0, E4 0} C_DIS
LIN {X -37.454, Y -96.835, Z 263.25, A 0, B 90, C 0, E1 0, E2 0, E3 0, E4 0} C_DIS
LIN {X -41.372, Y -97.687, Z 263.25, A 0, B 90, C 0, E1 0, E2 0, E3 0, E4 0} C_DIS
LIN {X -45.293, Y -98.518, Z 263.25, A 0, B 90, C 0, E1 0, E2 0, E3 0, E4 0} C_DIS
LIN {X -49.233, Y -99.257, Z 263.25, A 0, B 90, C 0, E1 0, E2 0, E3 0, E4 0} C_DIS
LIN {X -53.203, Y -99.813, Z 263.25, A 0, B 90, C 0, E1 0, E2 0, E3 0, E4 0} C_DIS
LIN {X -57.201, Y -100.081, Z 263.25, A 0, B 90, C 0, E1 0, E2 0, E3 0, E4 0} C_DIS
LIN {X -61.204, Y -99.928, Z 263.25, A 0, B 90, C 0, E1 0, E2 0, E3 0, E4 0} C_DIS
LIN {X -65.142, Y -99.201, Z 263.25, A 0, B 90, C 0, E1 0, E2 0, E3 0, E4 0} C_DIS
LIN {X -68.881, Y -97.773, Z 263.25, A 0, B 90, C 0, E1 0, E2 0, E3 0, E4 0} C_DIS
LIN {X -72.254, Y -95.62, Z 263.25, A 0, B 90, C 0, E1 0, E2 0, E3 0, E4 0} C_DIS
LIN {X -75.148, Y -92.854, Z 263.25, A 0, B 90, C 0, E1 0, E2 0, E3 0, E4 0} C_DIS
LIN {X -77.553, Y -89.651, Z 263.25, A 0, B 90, C 0, E1 0, E2 0, E3 0, E4 0} C_DIS
LIN {X -79.527, Y -86.165, Z 263.25, A 0, B 90, C 0, E1 0, E2 0, E3 0, E4 0} C_DIS
LIN {X -81.152, Y -82.501, Z 263.25, A 0, B 90, C 0, E1 0, E2 0, E3 0, E4 0} C_DIS
LIN {X -82.512, Y -78.731, Z 263.25, A 0, B 90, C 0, E1 0, E2 0, E3 0, E4 0} C_DIS
LIN {X -83.692, Y -74.9, Z 263.25, A 0, B 90, C 0, E1 0, E2 0, E3 0, E4 0} C_DIS
LIN {X -84.787, Y -71.043, Z 263.25, A 0, B 90, C 0, E1 0, E2 0, E3 0, E4 0} C_DIS
LIN {X -85.921, Y -67.199, Z 263.25, A 0, B 90, C 0, E1 0, E2 0, E3 0, E4 0} C_DIS
LIN {X -87.287, Y -63.432, Z 263.25, A 0, B 90, C 0, E1 0, E2 0, E3 0, E4 0} C_DIS
LIN {X -89.165, Y -59.897, Z 263.25, A 0, B 90, C 0, E1 0, E2 0, E3 0, E4 0} C_DIS
LIN {X -91.754, Y -56.847, Z 263.25, A 0, B 90, C 0, E1 0, E2 0, E3 0, E4 0} C_DIS
LIN {X -94.889, Y -54.356, Z 263.25, A 0, B 90, C 0, E1 0, E2 0, E3 0, E4 0} C_DIS
LIN {X -98.278, Y -52.215, Z 263.25, A 0, B 90, C 0, E1 0, E2 0, E3 0, E4 0} C_DIS
LIN {X -101.746, Y -50.205, Z 263.25, A 0, B 90, C 0, E1 0, E2 0, E3 0, E4 0} C_DIS
LIN {X -105.207, Y -48.182, Z 263.25, A 0, B 90, C 0, E1 0, E2 0, E3 0, E4 0} C_DIS
LIN {X -108.603, Y -46.052, Z 263.25, A 0, B 90, C 0, E1 0, E2 0, E3 0, E4 0} C_DIS
LIN {X -111.885, Y -43.751, Z 263.25, A 0, B 90, C 0, E1 0, E2 0, E3 0, E4 0} C_DIS
LIN {X -114.997, Y -41.226, Z 263.25, A 0, B 90, C 0, E1 0, E2 0, E3 0, E4 0} C_DIS
LIN {X -117.867, Y -38.429, Z 263.25, A 0, B 90, C 0, E1 0, E2 0, E3 0, E4 0} C_DIS
LIN {X -120.394, Y -35.322, Z 263.25, A 0, B 90, C 0, E1 0, E2 0, E3 0, E4 0} C_DIS
LIN {X -122.441, Y -31.88, Z 263.25, A 0, B 90, C 0, E1 0, E2 0, E3 0, E4 0} C_DIS
LIN {X -123.833, Y -28.128, Z 263.25, A 0, B 90, C 0, E1 0, E2 0, E3 0, E4 0} C_DIS
LIN {X -124.411, Y -24.169, Z 263.25, A 0, B 90, C 0, E1 0, E2 0, E3 0, E4 0} C_DIS
LIN {X -124.132, Y -20.177, Z 263.25, A 0, B 90, C 0, E1 0, E2 0, E3 0, E4 0} C_DIS
LIN {X -123.098, Y -16.309, Z 263.25, A 0, B 90, C 0, E1 0, E2 0, E3 0, E4 0} C_DIS
LIN {X -121.482, Y -12.643, Z 263.25, A 0, B 90, C 0, E1 0, E2 0, E3 0, E4 0} C_DIS
LIN {X -119.442, Y -9.195, Z 263.25, A 0, B 90, C 0, E1 0, E2 0, E3 0, E4 0} C_DIS
LIN {X -117.095, Y -5.947, Z 263.25, A 0, B 90, C 0, E1 0, E2 0, E3 0, E4 0} C_DIS
LIN {X -114.518, Y -2.879, Z 263.25, A 0, B 90, C 0, E1 0, E2 0, E3 0, E4 0} C_DIS
LIN {X -112.697, Y 0, Z 265.75, A 0, B 90, C 0, E1 0, E2 0, E3 0, E4 0} C_DIS
LIN {X -109.837, Y 2.55, Z 265.75, A 0, B 90, C 0, E1 0, E2 0, E3 0, E4 0} C_DIS
LIN {X -106.948, Y 5.391, Z 265.75, A 0, B 90, C 0, E1 0, E2 0, E3 0, E4 0} C_DIS
LIN {X -104.081, Y 8.256, Z 265.75, A 0, B 90, C 0, E1 0, E2 0, E3 0, E4 0} C_DIS
LIN {X -101.306, Y 11.21, Z 265.75, A 0, B 90, C 0, E1 0, E2 0, E3 0, E4 0} C_DIS
LIN {X -98.789, Y 14.383, Z 265.75, A 0, B 90, C 0, E1 0, E2 0, E3 0, E4 0} C_DIS
LIN {X -96.852, Y 17.934, Z 265.75, A 0, B 90, C 0, E1 0, E2 0, E3 0, E4 0} C_DIS
LIN {X -95.865, Y 21.853, Z 265.75, A 0, B 90, C 0, E1 0, E2 0, E3 0, E4 0} C_DIS
LIN {X -95.786, Y 25.9, Z 265.75, A 0, B 90, C 0, E1 0, E2 0, E3 0, E4 0} C_DIS
LIN {X -96.255, Y 29.925, Z 265.75, A 0, B 90, C 0, E1 0, E2 0, E3 0, E4 0} C_DIS
LIN {X -97.001, Y 33.908, Z 265.75, A 0, B 90, C 0, E1 0, E2 0, E3 0, E4 0} C_DIS
LIN {X -97.877, Y 37.866, Z 265.75, A 0, B 90, C 0, E1 0, E2 0, E3 0, E4 0} C_DIS
LIN {X -98.793, Y 41.814, Z 265.75, A 0, B 90, C 0, E1 0, E2 0, E3 0, E4 0} C_DIS
LIN {X -99.678, Y 45.769, Z 265.75, A 0, B 90, C 0, E1 0, E2 0, E3 0, E4 0} C_DIS
LIN {X -100.458, Y 49.747, Z 265.75, A 0, B 90, C 0, E1 0, E2 0, E3 0, E4 0} C_DIS
LIN {X -101.041, Y 53.757, Z 265.75, A 0, B 90, C 0, E1 0, E2 0, E3 0, E4 0} C_DIS
LIN {X -101.319, Y 57.799, Z 265.75, A 0, B 90, C 0, E1 0, E2 0, E3 0, E4 0} C_DIS
LIN {X -101.155, Y 61.847, Z 265.75, A 0, B 90, C 0, E1 0, E2 0, E3 0, E4 0} C_DIS
LIN {X -100.391, Y 65.822, Z 265.75, A 0, B 90, C 0, E1 0, E2 0, E3 0, E4 0} C_DIS
LIN {X -98.899, Y 69.583, Z 265.75, A 0, B 90, C 0, E1 0, E2 0, E3 0, E4 0} C_DIS
LIN {X -96.661, Y 72.954, Z 265.75, A 0, B 90, C 0, E1 0, E2 0, E3 0, E4 0} C_DIS
LIN {X -93.803, Y 75.819, Z 265.75, A 0, B 90, C 0, E1 0, E2 0, E3 0, E4 0} C_DIS
LIN {X -90.508, Y 78.173, Z 265.75, A 0, B 90, C 0, E1 0, E2 0, E3 0, E4 0} C_DIS
LIN {X -86.934, Y 80.082, Z 265.75, A 0, B 90, C 0, E1 0, E2 0, E3 0, E4 0} C_DIS
LIN {X -83.19, Y 81.631, Z 265.75, A 0, B 90, C 0, E1 0, E2 0, E3 0, E4 0} C_DIS
LIN {X -79.345, Y 82.911, Z 265.75, A 0, B 90, C 0, E1 0, E2 0, E3 0, E4 0} C_DIS
LIN {X -75.444, Y 84.01, Z 265.75, A 0, B 90, C 0, E1 0, E2 0, E3 0, E4 0} C_DIS
LIN {X -71.52, Y 85.025, Z 265.75, A 0, B 90, C 0, E1 0, E2 0, E3 0, E4 0} C_DIS
LIN {X -67.608, Y 86.086, Z 265.75, A 0, B 90, C 0, E1 0, E2 0, E3 0, E4 0} C_DIS
LIN {X -63.772, Y 87.39, Z 265.75, A 0, B 90, C 0, E1 0, E2 0, E3 0, E4 0} C_DIS
LIN {X -60.166, Y 89.228, Z 265.75, A 0, B 90, C 0, E1 0, E2 0, E3 0, E4 0} C_DIS
LIN {X -57.056, Y 91.812, Z 265.75, A 0, B 90, C 0, E1 0, E2 0, E3 0, E4 0} C_DIS
LIN {X -54.532, Y 94.978, Z 265.75, A 0, B 90, C 0, E1 0, E2 0, E3 0, E4 0} C_DIS
LIN {X -52.384, Y 98.414, Z 265.75, A 0, B 90, C 0, E1 0, E2 0, E3 0, E4 0} C_DIS
LIN {X -50.384, Y 101.94, Z 265.75, A 0, B 90, C 0, E1 0, E2 0, E3 0, E4 0} C_DIS
LIN {X -48.381, Y 105.463, Z 265.75, A 0, B 90, C 0, E1 0, E2 0, E3 0, E4 0} C_DIS
LIN {X -46.278, Y 108.928, Z 265.75, A 0, B 90, C 0, E1 0, E2 0, E3 0, E4 0} C_DIS
LIN {X -44.006, Y 112.283, Z 265.75, A 0, B 90, C 0, E1 0, E2 0, E3 0, E4 0} C_DIS
LIN {X -41.508, Y 115.474, Z 265.75, A 0, B 90, C 0, E1 0, E2 0, E3 0, E4 0} C_DIS
LIN {X -38.736, Y 118.429, Z 265.75, A 0, B 90, C 0, E1 0, E2 0, E3 0, E4 0} C_DIS
LIN {X -35.644, Y 121.045, Z 265.75, A 0, B 90, C 0, E1 0, E2 0, E3 0, E4 0} C_DIS
LIN {X -32.205, Y 123.182, Z 265.75, A 0, B 90, C 0, E1 0, E2 0, E3 0, E4 0} C_DIS
LIN {X -28.436, Y 124.656, Z 265.75, A 0, B 90, C 0, E1 0, E2 0, E3 0, E4 0} C_DIS
LIN {X -24.443, Y 125.301, Z 265.75, A 0, B 90, C 0, E1 0, E2 0, E3 0, E4 0} C_DIS
LIN {X -20.405, Y 125.063, Z 265.75, A 0, B 90, C 0, E1 0, E2 0, E3 0, E4 0} C_DIS
LIN {X -16.487, Y 124.044, Z 265.75, A 0, B 90, C 0, E1 0, E2 0, E3 0, E4 0} C_DIS
LIN {X -12.775, Y 122.423, Z 265.75, A 0, B 90, C 0, E1 0, E2 0, E3 0, E4 0} C_DIS
LIN {X -9.286, Y 120.364, Z 265.75, A 0, B 90, C 0, E1 0, E2 0, E3 0, E4 0} C_DIS
LIN {X -6.004, Y 117.988, Z 265.75, A 0, B 90, C 0, E1 0, E2 0, E3 0, E4 0} C_DIS
LIN {X -2.906, Y 115.378, Z 265.75, A 0, B 90, C 0, E1 0, E2 0, E3 0, E4 0} C_DIS
LIN {X 0, Y 112.697, Z 265.75, A 0, B 90, C 0, E1 0, E2 0, E3 0, E4 0} C_DIS
LIN {X 2.55, Y 109.837, Z 265.75, A 0, B 90, C 0, E1 0, E2 0, E3 0, E4 0} C_DIS
LIN {X 5.391, Y 106.948, Z 265.75, A 0, B 90, C 0, E1 0, E2 0, E3 0, E4 0} C_DIS
LIN {X 8.256, Y 104.081, Z 265.75, A 0, B 90, C 0, E1 0, E2 0, E3 0, E4 0} C_DIS
LIN {X 11.21, Y 101.306, Z 265.75, A 0, B 90, C 0, E1 0, E2 0, E3 0, E4 0} C_DIS
LIN {X 14.383, Y 98.789, Z 265.75, A 0, B 90, C 0, E1 0, E2 0, E3 0, E4 0} C_DIS
LIN {X 17.934, Y 96.852, Z 265.75, A 0, B 90, C 0, E1 0, E2 0, E3 0, E4 0} C_DIS
LIN {X 21.853, Y 95.865, Z 265.75, A 0, B 90, C 0, E1 0, E2 0, E3 0, E4 0} C_DIS
LIN {X 25.9, Y 95.786, Z 265.75, A 0, B 90, C 0, E1 0, E2 0, E3 0, E4 0} C_DIS
LIN {X 29.925, Y 96.255, Z 265.75, A 0, B 90, C 0, E1 0, E2 0, E3 0, E4 0} C_DIS
LIN {X 33.908, Y 97.001, Z 265.75, A 0, B 90, C 0, E1 0, E2 0, E3 0, E4 0} C_DIS
LIN {X 37.866, Y 97.877, Z 265.75, A 0, B 90, C 0, E1 0, E2 0, E3 0, E4 0} C_DIS
LIN {X 41.814, Y 98.793, Z 265.75, A 0, B 90, C 0, E1 0, E2 0, E3 0, E4 0} C_DIS
LIN {X 45.769, Y 99.678, Z 265.75, A 0, B 90, C 0, E1 0, E2 0, E3 0, E4 0} C_DIS
LIN {X 49.747, Y 100.458, Z 265.75, A 0, B 90, C 0, E1 0, E2 0, E3 0, E4 0} C_DIS
LIN {X 53.757, Y 101.041, Z 265.75, A 0, B 90, C 0, E1 0, E2 0, E3 0, E4 0} C_DIS
LIN {X 57.799, Y 101.319, Z 265.75, A 0, B 90, C 0, E1 0, E2 0, E3 0, E4 0} C_DIS
LIN {X 61.847, Y 101.155, Z 265.75, A 0, B 90, C 0, E1 0, E2 0, E3 0, E4 0} C_DIS
LIN {X 65.822, Y 100.391, Z 265.75, A 0, B 90, C 0, E1 0, E2 0, E3 0, E4 0} C_DIS
LIN {X 69.583, Y 98.899, Z 265.75, A 0, B 90, C 0, E1 0, E2 0, E3 0, E4 0} C_DIS
LIN {X 72.954, Y 96.661, Z 265.75, A 0, B 90, C 0, E1 0, E2 0, E3 0, E4 0} C_DIS
LIN {X 75.819, Y 93.803, Z 265.75, A 0, B 90, C 0, E1 0, E2 0, E3 0, E4 0} C_DIS
LIN {X 78.173, Y 90.508, Z 265.75, A 0, B 90, C 0, E1 0, E2 0, E3 0, E4 0} C_DIS
LIN {X 80.082, Y 86.934, Z 265.75, A 0, B 90, C 0, E1 0, E2 0, E3 0, E4 0} C_DIS
LIN {X 81.631, Y 83.19, Z 265.75, A 0, B 90, C 0, E1 0, E2 0, E3 0, E4 0} C_DIS
LIN {X 82.911, Y 79.345, Z 265.75, A 0, B 90, C 0, E1 0, E2 0, E3 0, E4 0} C_DIS
LIN {X 84.01, Y 75.444, Z 265.75, A 0, B 90, C 0, E1 0, E2 0, E3 0, E4 0} C_DIS
LIN {X 85.025, Y 71.52, Z 265.75, A 0, B 90, C 0, E1 0, E2 0, E3 0, E4 0} C_DIS
LIN {X 86.086, Y 67.608, Z 265.75, A 0, B 90, C 0, E1 0, E2 0, E3 0, E4 0} C_DIS
LIN {X 87.39, Y 63.772, Z 265.75, A 0, B 90, C 0, E1 0, E2 0, E3 0, E4 0} C_DIS
LIN {X 89.228, Y 60.166, Z 265.75, A 0, B 90, C 0, E1 0, E2 0, E3 0, E4 0} C_DIS
LIN {X 91.812, Y 57.056, Z 265.75, A 0, B 90, C 0, E1 0, E2 0, E3 0, E4 0} C_DIS
LIN {X 94.978, Y 54.532, Z 265.75, A 0, B 90, C 0, E1 0, E2 0, E3 0, E4 0} C_DIS
LIN {X 98.414, Y 52.384, Z 265.75, A 0, B 90, C 0, E1 0, E2 0, E3 0, E4 0} C_DIS
LIN {X 101.94, Y 50.384, Z 265.75, A 0, B 90, C 0, E1 0, E2 0, E3 0, E4 0} C_DIS
LIN {X 105.463, Y 48.381, Z 265.75, A 0, B 90, C 0, E1 0, E2 0, E3 0, E4 0} C_DIS
LIN {X 108.928, Y 46.278, Z 265.75, A 0, B 90, C 0, E1 0, E2 0, E3 0, E4 0} C_DIS
LIN {X 112.283, Y 44.006, Z 265.75, A 0, B 90, C 0, E1 0, E2 0, E3 0, E4 0} C_DIS
LIN {X 115.474, Y 41.508, Z 265.75, A 0, B 90, C 0, E1 0, E2 0, E3 0, E4 0} C_DIS
LIN {X 118.429, Y 38.736, Z 265.75, A 0, B 90, C 0, E1 0, E2 0, E3 0, E4 0} C_DIS
LIN {X 121.045, Y 35.644, Z 265.75, A 0, B 90, C 0, E1 0, E2 0, E3 0, E4 0} C_DIS
LIN {X 123.182, Y 32.205, Z 265.75, A 0, B 90, C 0, E1 0, E2 0, E3 0, E4 0} C_DIS
LIN {X 124.656, Y 28.436, Z 265.75, A 0, B 90, C 0, E1 0, E2 0, E3 0, E4 0} C_DIS
LIN {X 125.301, Y 24.443, Z 265.75, A 0, B 90, C 0, E1 0, E2 0, E3 0, E4 0} C_DIS
LIN {X 125.063, Y 20.405, Z 265.75, A 0, B 90, C 0, E1 0, E2 0, E3 0, E4 0} C_DIS
LIN {X 124.044, Y 16.487, Z 265.75, A 0, B 90, C 0, E1 0, E2 0, E3 0, E4 0} C_DIS
LIN {X 122.423, Y 12.775, Z 265.75, A 0, B 90, C 0, E1 0, E2 0, E3 0, E4 0} C_DIS
LIN {X 120.364, Y 9.286, Z 265.75, A 0, B 90, C 0, E1 0, E2 0, E3 0, E4 0} C_DIS
LIN {X 117.988, Y 6.004, Z 265.75, A 0, B 90, C 0, E1 0, E2 0, E3 0, E4 0} C_DIS
LIN {X 115.378, Y 2.906, Z 265.75, A 0, B 90, C 0, E1 0, E2 0, E3 0, E4 0} C_DIS
LIN {X 112.697, Y 0, Z 265.75, A 0, B 90, C 0, E1 0, E2 0, E3 0, E4 0} C_DIS
LIN {X 109.837, Y -2.55, Z 265.75, A 0, B 90, C 0, E1 0, E2 0, E3 0, E4 0} C_DIS
LIN {X 106.948, Y -5.391, Z 265.75, A 0, B 90, C 0, E1 0, E2 0, E3 0, E4 0} C_DIS
LIN {X 104.081, Y -8.256, Z 265.75, A 0, B 90, C 0, E1 0, E2 0, E3 0, E4 0} C_DIS
LIN {X 101.306, Y -11.21, Z 265.75, A 0, B 90, C 0, E1 0, E2 0, E3 0, E4 0} C_DIS
LIN {X 98.789, Y -14.383, Z 265.75, A 0, B 90, C 0, E1 0, E2 0, E3 0, E4 0} C_DIS
LIN {X 96.852, Y -17.934, Z 265.75, A 0, B 90, C 0, E1 0, E2 0, E3 0, E4 0} C_DIS
LIN {X 95.865, Y -21.853, Z 265.75, A 0, B 90, C 0, E1 0, E2 0, E3 0, E4 0} C_DIS
LIN {X 95.786, Y -25.9, Z 265.75, A 0, B 90, C 0, E1 0, E2 0, E3 0, E4 0} C_DIS
LIN {X 96.255, Y -29.925, Z 265.75, A 0, B 90, C 0, E1 0, E2 0, E3 0, E4 0} C_DIS
LIN {X 97.001, Y -33.908, Z 265.75, A 0, B 90, C 0, E1 0, E2 0, E3 0, E4 0} C_DIS
LIN {X 97.877, Y -37.866, Z 265.75, A 0, B 90, C 0, E1 0, E2 0, E3 0, E4 0} C_DIS
LIN {X 98.793, Y -41.814, Z 265.75, A 0, B 90, C 0, E1 0, E2 0, E3 0, E4 0} C_DIS
LIN {X 99.678, Y -45.769, Z 265.75, A 0, B 90, C 0, E1 0, E2 0, E3 0, E4 0} C_DIS
LIN {X 100.458, Y -49.747, Z 265.75, A 0, B 90, C 0, E1 0, E2 0, E3 0, E4 0} C_DIS
LIN {X 101.041, Y -53.757, Z 265.75, A 0, B 90, C 0, E1 0, E2 0, E3 0, E4 0} C_DIS
LIN {X 101.319, Y -57.799, Z 265.75, A 0, B 90, C 0, E1 0, E2 0, E3 0, E4 0} C_DIS
LIN {X 101.155, Y -61.847, Z 265.75, A 0, B 90, C 0, E1 0, E2 0, E3 0, E4 0} C_DIS
LIN {X 100.391, Y -65.822, Z 265.75, A 0, B 90, C 0, E1 0, E2 0, E3 0, E4 0} C_DIS
LIN {X 98.899, Y -69.583, Z 265.75, A 0, B 90, C 0, E1 0, E2 0, E3 0, E4 0} C_DIS
LIN {X 96.661, Y -72.954, Z 265.75, A 0, B 90, C 0, E1 0, E2 0, E3 0, E4 0} C_DIS
LIN {X 93.803, Y -75.819, Z 265.75, A 0, B 90, C 0, E1 0, E2 0, E3 0, E4 0} C_DIS
LIN {X 90.508, Y -78.173, Z 265.75, A 0, B 90, C 0, E1 0, E2 0, E3 0, E4 0} C_DIS
LIN {X 86.934, Y -80.082, Z 265.75, A 0, B 90, C 0, E1 0, E2 0, E3 0, E4 0} C_DIS
LIN {X 83.19, Y -81.631, Z 265.75, A 0, B 90, C 0, E1 0, E2 0, E3 0, E4 0} C_DIS
LIN {X 79.345, Y -82.911, Z 265.75, A 0, B 90, C 0, E1 0, E2 0, E3 0, E4 0} C_DIS
LIN {X 75.444, Y -84.01, Z 265.75, A 0, B 90, C 0, E1 0, E2 0, E3 0, E4 0} C_DIS
LIN {X 71.52, Y -85.025, Z 265.75, A 0, B 90, C 0, E1 0, E2 0, E3 0, E4 0} C_DIS
LIN {X 67.608, Y -86.086, Z 265.75, A 0, B 90, C 0, E1 0, E2 0, E3 0, E4 0} C_DIS
LIN {X 63.772, Y -87.39, Z 265.75, A 0, B 90, C 0, E1 0, E2 0, E3 0, E4 0} C_DIS
LIN {X 60.166, Y -89.228, Z 265.75, A 0, B 90, C 0, E1 0, E2 0, E3 0, E4 0} C_DIS
LIN {X 57.056, Y -91.812, Z 265.75, A 0, B 90, C 0, E1 0, E2 0, E3 0, E4 0} C_DIS
LIN {X 54.532, Y -94.978, Z 265.75, A 0, B 90, C 0, E1 0, E2 0, E3 0, E4 0} C_DIS
LIN {X 52.384, Y -98.414, Z 265.75, A 0, B 90, C 0, E1 0, E2 0, E3 0, E4 0} C_DIS
LIN {X 50.384, Y -101.94, Z 265.75, A 0, B 90, C 0, E1 0, E2 0, E3 0, E4 0} C_DIS
LIN {X 48.381, Y -105.463, Z 265.75, A 0, B 90, C 0, E1 0, E2 0, E3 0, E4 0} C_DIS
LIN {X 46.278, Y -108.928, Z 265.75, A 0, B 90, C 0, E1 0, E2 0, E3 0, E4 0} C_DIS
LIN {X 44.006, Y -112.283, Z 265.75, A 0, B 90, C 0, E1 0, E2 0, E3 0, E4 0} C_DIS
LIN {X 41.508, Y -115.474, Z 265.75, A 0, B 90, C 0, E1 0, E2 0, E3 0, E4 0} C_DIS
LIN {X 38.736, Y -118.429, Z 265.75, A 0, B 90, C 0, E1 0, E2 0, E3 0, E4 0} C_DIS
LIN {X 35.644, Y -121.045, Z 265.75, A 0, B 90, C 0, E1 0, E2 0, E3 0, E4 0} C_DIS
LIN {X 32.205, Y -123.182, Z 265.75, A 0, B 90, C 0, E1 0, E2 0, E3 0, E4 0} C_DIS
LIN {X 28.436, Y -124.656, Z 265.75, A 0, B 90, C 0, E1 0, E2 0, E3 0, E4 0} C_DIS
LIN {X 24.443, Y -125.301, Z 265.75, A 0, B 90, C 0, E1 0, E2 0, E3 0, E4 0} C_DIS
LIN {X 20.405, Y -125.063, Z 265.75, A 0, B 90, C 0, E1 0, E2 0, E3 0, E4 0} C_DIS
LIN {X 16.487, Y -124.044, Z 265.75, A 0, B 90, C 0, E1 0, E2 0, E3 0, E4 0} C_DIS
LIN {X 12.775, Y -122.423, Z 265.75, A 0, B 90, C 0, E1 0, E2 0, E3 0, E4 0} C_DIS
LIN {X 9.286, Y -120.364, Z 265.75, A 0, B 90, C 0, E1 0, E2 0, E3 0, E4 0} C_DIS
LIN {X 6.004, Y -117.988, Z 265.75, A 0, B 90, C 0, E1 0, E2 0, E3 0, E4 0} C_DIS
LIN {X 2.906, Y -115.378, Z 265.75, A 0, B 90, C 0, E1 0, E2 0, E3 0, E4 0} C_DIS
LIN {X 0, Y -112.697, Z 265.75, A 0, B 90, C 0, E1 0, E2 0, E3 0, E4 0} C_DIS
LIN {X -2.55, Y -109.837, Z 265.75, A 0, B 90, C 0, E1 0, E2 0, E3 0, E4 0} C_DIS
LIN {X -5.391, Y -106.948, Z 265.75, A 0, B 90, C 0, E1 0, E2 0, E3 0, E4 0} C_DIS
LIN {X -8.256, Y -104.081, Z 265.75, A 0, B 90, C 0, E1 0, E2 0, E3 0, E4 0} C_DIS
LIN {X -11.21, Y -101.306, Z 265.75, A 0, B 90, C 0, E1 0, E2 0, E3 0, E4 0} C_DIS
LIN {X -14.383, Y -98.789, Z 265.75, A 0, B 90, C 0, E1 0, E2 0, E3 0, E4 0} C_DIS
LIN {X -17.934, Y -96.852, Z 265.75, A 0, B 90, C 0, E1 0, E2 0, E3 0, E4 0} C_DIS
LIN {X -21.853, Y -95.865, Z 265.75, A 0, B 90, C 0, E1 0, E2 0, E3 0, E4 0} C_DIS
LIN {X -25.9, Y -95.786, Z 265.75, A 0, B 90, C 0, E1 0, E2 0, E3 0, E4 0} C_DIS
LIN {X -29.925, Y -96.255, Z 265.75, A 0, B 90, C 0, E1 0, E2 0, E3 0, E4 0} C_DIS
LIN {X -33.908, Y -97.001, Z 265.75, A 0, B 90, C 0, E1 0, E2 0, E3 0, E4 0} C_DIS
LIN {X -37.866, Y -97.877, Z 265.75, A 0, B 90, C 0, E1 0, E2 0, E3 0, E4 0} C_DIS
LIN {X -41.814, Y -98.793, Z 265.75, A 0, B 90, C 0, E1 0, E2 0, E3 0, E4 0} C_DIS
LIN {X -45.769, Y -99.678, Z 265.75, A 0, B 90, C 0, E1 0, E2 0, E3 0, E4 0} C_DIS
LIN {X -49.747, Y -100.458, Z 265.75, A 0, B 90, C 0, E1 0, E2 0, E3 0, E4 0} C_DIS
LIN {X -53.757, Y -101.041, Z 265.75, A 0, B 90, C 0, E1 0, E2 0, E3 0, E4 0} C_DIS
LIN {X -57.799, Y -101.319, Z 265.75, A 0, B 90, C 0, E1 0, E2 0, E3 0, E4 0} C_DIS
LIN {X -61.847, Y -101.155, Z 265.75, A 0, B 90, C 0, E1 0, E2 0, E3 0, E4 0} C_DIS
LIN {X -65.822, Y -100.391, Z 265.75, A 0, B 90, C 0, E1 0, E2 0, E3 0, E4 0} C_DIS
LIN {X -69.583, Y -98.899, Z 265.75, A 0, B 90, C 0, E1 0, E2 0, E3 0, E4 0} C_DIS
LIN {X -72.954, Y -96.661, Z 265.75, A 0, B 90, C 0, E1 0, E2 0, E3 0, E4 0} C_DIS
LIN {X -75.819, Y -93.803, Z 265.75, A 0, B 90, C 0, E1 0, E2 0, E3 0, E4 0} C_DIS
LIN {X -78.173, Y -90.508, Z 265.75, A 0, B 90, C 0, E1 0, E2 0, E3 0, E4 0} C_DIS
LIN {X -80.082, Y -86.934, Z 265.75, A 0, B 90, C 0, E1 0, E2 0, E3 0, E4 0} C_DIS
LIN {X -81.631, Y -83.19, Z 265.75, A 0, B 90, C 0, E1 0, E2 0, E3 0, E4 0} C_DIS
LIN {X -82.911, Y -79.345, Z 265.75, A 0, B 90, C 0, E1 0, E2 0, E3 0, E4 0} C_DIS
LIN {X -84.01, Y -75.444, Z 265.75, A 0, B 90, C 0, E1 0, E2 0, E3 0, E4 0} C_DIS
LIN {X -85.025, Y -71.52, Z 265.75, A 0, B 90, C 0, E1 0, E2 0, E3 0, E4 0} C_DIS
LIN {X -86.086, Y -67.608, Z 265.75, A 0, B 90, C 0, E1 0, E2 0, E3 0, E4 0} C_DIS
LIN {X -87.39, Y -63.772, Z 265.75, A 0, B 90, C 0, E1 0, E2 0, E3 0, E4 0} C_DIS
LIN {X -89.228, Y -60.166, Z 265.75, A 0, B 90, C 0, E1 0, E2 0, E3 0, E4 0} C_DIS
LIN {X -91.812, Y -57.056, Z 265.75, A 0, B 90, C 0, E1 0, E2 0, E3 0, E4 0} C_DIS
LIN {X -94.978, Y -54.532, Z 265.75, A 0, B 90, C 0, E1 0, E2 0, E3 0, E4 0} C_DIS
LIN {X -98.414, Y -52.384, Z 265.75, A 0, B 90, C 0, E1 0, E2 0, E3 0, E4 0} C_DIS
LIN {X -101.94, Y -50.384, Z 265.75, A 0, B 90, C 0, E1 0, E2 0, E3 0, E4 0} C_DIS
LIN {X -105.463, Y -48.381, Z 265.75, A 0, B 90, C 0, E1 0, E2 0, E3 0, E4 0} C_DIS
LIN {X -108.928, Y -46.278, Z 265.75, A 0, B 90, C 0, E1 0, E2 0, E3 0, E4 0} C_DIS
LIN {X -112.283, Y -44.006, Z 265.75, A 0, B 90, C 0, E1 0, E2 0, E3 0, E4 0} C_DIS
LIN {X -115.474, Y -41.508, Z 265.75, A 0, B 90, C 0, E1 0, E2 0, E3 0, E4 0} C_DIS
LIN {X -118.429, Y -38.736, Z 265.75, A 0, B 90, C 0, E1 0, E2 0, E3 0, E4 0} C_DIS
LIN {X -121.045, Y -35.644, Z 265.75, A 0, B 90, C 0, E1 0, E2 0, E3 0, E4 0} C_DIS
LIN {X -123.182, Y -32.205, Z 265.75, A 0, B 90, C 0, E1 0, E2 0, E3 0, E4 0} C_DIS
LIN {X -124.656, Y -28.436, Z 265.75, A 0, B 90, C 0, E1 0, E2 0, E3 0, E4 0} C_DIS
LIN {X -125.301, Y -24.443, Z 265.75, A 0, B 90, C 0, E1 0, E2 0, E3 0, E4 0} C_DIS
LIN {X -125.063, Y -20.405, Z 265.75, A 0, B 90, C 0, E1 0, E2 0, E3 0, E4 0} C_DIS
LIN {X -124.044, Y -16.487, Z 265.75, A 0, B 90, C 0, E1 0, E2 0, E3 0, E4 0} C_DIS
LIN {X -122.423, Y -12.775, Z 265.75, A 0, B 90, C 0, E1 0, E2 0, E3 0, E4 0} C_DIS
LIN {X -120.364, Y -9.286, Z 265.75, A 0, B 90, C 0, E1 0, E2 0, E3 0, E4 0} C_DIS
LIN {X -117.988, Y -6.004, Z 265.75, A 0, B 90, C 0, E1 0, E2 0, E3 0, E4 0} C_DIS
LIN {X -115.378, Y -2.906, Z 265.75, A 0, B 90, C 0, E1 0, E2 0, E3 0, E4 0} C_DIS
LIN {X -113.532, Y 0, Z 268.25, A 0, B 90, C 0, E1 0, E2 0, E3 0, E4 0} C_DIS
LIN {X -110.633, Y 2.58, Z 268.25, A 0, B 90, C 0, E1 0, E2 0, E3 0, E4 0} C_DIS
LIN {X -107.706, Y 5.447, Z 268.25, A 0, B 90, C 0, E1 0, E2 0, E3 0, E4 0} C_DIS
LIN {X -104.801, Y 8.339, Z 268.25, A 0, B 90, C 0, E1 0, E2 0, E3 0, E4 0} C_DIS
LIN {X -101.995, Y 11.326, Z 268.25, A 0, B 90, C 0, E1 0, E2 0, E3 0, E4 0} C_DIS
LIN {X -99.46, Y 14.543, Z 268.25, A 0, B 90, C 0, E1 0, E2 0, E3 0, E4 0} C_DIS
LIN {X -97.535, Y 18.152, Z 268.25, A 0, B 90, C 0, E1 0, E2 0, E3 0, E4 0} C_DIS
LIN {X -96.601, Y 22.13, Z 268.25, A 0, B 90, C 0, E1 0, E2 0, E3 0, E4 0} C_DIS
LIN {X -96.601, Y 26.223, Z 268.25, A 0, B 90, C 0, E1 0, E2 0, E3 0, E4 0} C_DIS
LIN {X -97.155, Y 30.283, Z 268.25, A 0, B 90, C 0, E1 0, E2 0, E3 0, E4 0} C_DIS
LIN {X -97.983, Y 34.297, Z 268.25, A 0, B 90, C 0, E1 0, E2 0, E3 0, E4 0} C_DIS
LIN {X -98.933, Y 38.284, Z 268.25, A 0, B 90, C 0, E1 0, E2 0, E3 0, E4 0} C_DIS
LIN {X -99.915, Y 42.263, Z 268.25, A 0, B 90, C 0, E1 0, E2 0, E3 0, E4 0} C_DIS
LIN {X -100.854, Y 46.253, Z 268.25, A 0, B 90, C 0, E1 0, E2 0, E3 0, E4 0} C_DIS
LIN {X -101.675, Y 50.268, Z 268.25, A 0, B 90, C 0, E1 0, E2 0, E3 0, E4 0} C_DIS
LIN {X -102.285, Y 54.321, Z 268.25, A 0, B 90, C 0, E1 0, E2 0, E3 0, E4 0} C_DIS
LIN {X -102.572, Y 58.408, Z 268.25, A 0, B 90, C 0, E1 0, E2 0, E3 0, E4 0} C_DIS
LIN {X -102.395, Y 62.5, Z 268.25, A 0, B 90, C 0, E1 0, E2 0, E3 0, E4 0} C_DIS
LIN {X -101.592, Y 66.514, Z 268.25, A 0, B 90, C 0, E1 0, E2 0, E3 0, E4 0} C_DIS
LIN {X -100.033, Y 70.297, Z 268.25, A 0, B 90, C 0, E1 0, E2 0, E3 0, E4 0} C_DIS
LIN {X -97.708, Y 73.663, Z 268.25, A 0, B 90, C 0, E1 0, E2 0, E3 0, E4 0} C_DIS
LIN {X -94.755, Y 76.497, Z 268.25, A 0, B 90, C 0, E1 0, E2 0, E3 0, E4 0} C_DIS
LIN {X -91.368, Y 78.799, Z 268.25, A 0, B 90, C 0, E1 0, E2 0, E3 0, E4 0} C_DIS
LIN {X -87.708, Y 80.639, Z 268.25, A 0, B 90, C 0, E1 0, E2 0, E3 0, E4 0} C_DIS
LIN {X -83.885, Y 82.113, Z 268.25, A 0, B 90, C 0, E1 0, E2 0, E3 0, E4 0} C_DIS
LIN {X -79.966, Y 83.313, Z 268.25, A 0, B 90, C 0, E1 0, E2 0, E3 0, E4 0} C_DIS
LIN {X -75.996, Y 84.33, Z 268.25, A 0, B 90, C 0, E1 0, E2 0, E3 0, E4 0} C_DIS
LIN {X -72.005, Y 85.266, Z 268.25, A 0, B 90, C 0, E1 0, E2 0, E3 0, E4 0} C_DIS
LIN {X -68.027, Y 86.253, Z 268.25, A 0, B 90, C 0, E1 0, E2 0, E3 0, E4 0} C_DIS
LIN {X -64.122, Y 87.492, Z 268.25, A 0, B 90, C 0, E1 0, E2 0, E3 0, E4 0} C_DIS
LIN {X -60.444, Y 89.286, Z 268.25, A 0, B 90, C 0, E1 0, E2 0, E3 0, E4 0} C_DIS
LIN {X -57.271, Y 91.864, Z 268.25, A 0, B 90, C 0, E1 0, E2 0, E3 0, E4 0} C_DIS
LIN {X -54.711, Y 95.059, Z 268.25, A 0, B 90, C 0, E1 0, E2 0, E3 0, E4 0} C_DIS
LIN {X -52.556, Y 98.544, Z 268.25, A 0, B 90, C 0, E1 0, E2 0, E3 0, E4 0} C_DIS
LIN {X -50.565, Y 102.127, Z 268.25, A 0, B 90, C 0, E1 0, E2 0, E3 0, E4 0} C_DIS
LIN {X -48.582, Y 105.714, Z 268.25, A 0, B 90, C 0, E1 0, E2 0, E3 0, E4 0} C_DIS
LIN {X -46.505, Y 109.248, Z 268.25, A 0, B 90, C 0, E1 0, E2 0, E3 0, E4 0} C_DIS
LIN {X -44.262, Y 112.678, Z 268.25, A 0, B 90, C 0, E1 0, E2 0, E3 0, E4 0} C_DIS
LIN {X -41.794, Y 115.948, Z 268.25, A 0, B 90, C 0, E1 0, E2 0, E3 0, E4 0} C_DIS
LIN {X -39.046, Y 118.988, Z 268.25, A 0, B 90, C 0, E1 0, E2 0, E3 0, E4 0} C_DIS
LIN {X -35.972, Y 121.694, Z 268.25, A 0, B 90, C 0, E1 0, E2 0, E3 0, E4 0} C_DIS
LIN {X -32.536, Y 123.922, Z 268.25, A 0, B 90, C 0, E1 0, E2 0, E3 0, E4 0} C_DIS
LIN {X -28.754, Y 125.482, Z 268.25, A 0, B 90, C 0, E1 0, E2 0, E3 0, E4 0} C_DIS
LIN {X -24.726, Y 126.196, Z 268.25, A 0, B 90, C 0, E1 0, E2 0, E3 0, E4 0} C_DIS
LIN {X -20.64, Y 126.002, Z 268.25, A 0, B 90, C 0, E1 0, E2 0, E3 0, E4 0} C_DIS
LIN {X -16.671, Y 125.001, Z 268.25, A 0, B 90, C 0, E1 0, E2 0, E3 0, E4 0} C_DIS
LIN {X -12.912, Y 123.375, Z 268.25, A 0, B 90, C 0, E1 0, E2 0, E3 0, E4 0} C_DIS
LIN {X -9.382, Y 121.297, Z 268.25, A 0, B 90, C 0, E1 0, E2 0, E3 0, E4 0} C_DIS
LIN {X -6.063, Y 118.893, Z 268.25, A 0, B 90, C 0, E1 0, E2 0, E3 0, E4 0} C_DIS
LIN {X -2.934, Y 116.25, Z 268.25, A 0, B 90, C 0, E1 0, E2 0, E3 0, E4 0} C_DIS
LIN {X 0, Y 113.532, Z 268.25, A 0, B 90, C 0, E1 0, E2 0, E3 0, E4 0} C_DIS
LIN {X 2.58, Y 110.633, Z 268.25, A 0, B 90, C 0, E1 0, E2 0, E3 0, E4 0} C_DIS
LIN {X 5.447, Y 107.706, Z 268.25, A 0, B 90, C 0, E1 0, E2 0, E3 0, E4 0} C_DIS
LIN {X 8.339, Y 104.801, Z 268.25, A 0, B 90, C 0, E1 0, E2 0, E3 0, E4 0} C_DIS
LIN {X 11.326, Y 101.995, Z 268.25, A 0, B 90, C 0, E1 0, E2 0, E3 0, E4 0} C_DIS
LIN {X 14.543, Y 99.46, Z 268.25, A 0, B 90, C 0, E1 0, E2 0, E3 0, E4 0} C_DIS
LIN {X 18.152, Y 97.535, Z 268.25, A 0, B 90, C 0, E1 0, E2 0, E3 0, E4 0} C_DIS
LIN {X 22.13, Y 96.601, Z 268.25, A 0, B 90, C 0, E1 0, E2 0, E3 0, E4 0} C_DIS
LIN {X 26.223, Y 96.601, Z 268.25, A 0, B 90, C 0, E1 0, E2 0, E3 0, E4 0} C_DIS
LIN {X 30.283, Y 97.155, Z 268.25, A 0, B 90, C 0, E1 0, E2 0, E3 0, E4 0} C_DIS
LIN {X 34.297, Y 97.983, Z 268.25, A 0, B 90, C 0, E1 0, E2 0, E3 0, E4 0} C_DIS
LIN {X 38.284, Y 98.933, Z 268.25, A 0, B 90, C 0, E1 0, E2 0, E3 0, E4 0} C_DIS
LIN {X 42.263, Y 99.915, Z 268.25, A 0, B 90, C 0, E1 0, E2 0, E3 0, E4 0} C_DIS
LIN {X 46.253, Y 100.854, Z 268.25, A 0, B 90, C 0, E1 0, E2 0, E3 0, E4 0} C_DIS
LIN {X 50.268, Y 101.675, Z 268.25, A 0, B 90, C 0, E1 0, E2 0, E3 0, E4 0} C_DIS
LIN {X 54.321, Y 102.285, Z 268.25, A 0, B 90, C 0, E1 0, E2 0, E3 0, E4 0} C_DIS
LIN {X 58.408, Y 102.572, Z 268.25, A 0, B 90, C 0, E1 0, E2 0, E3 0, E4 0} C_DIS
LIN {X 62.5, Y 102.395, Z 268.25, A 0, B 90, C 0, E1 0, E2 0, E3 0, E4 0} C_DIS
LIN {X 66.514, Y 101.592, Z 268.25, A 0, B 90, C 0, E1 0, E2 0, E3 0, E4 0} C_DIS
LIN {X 70.297, Y 100.033, Z 268.25, A 0, B 90, C 0, E1 0, E2 0, E3 0, E4 0} C_DIS
LIN {X 73.663, Y 97.708, Z 268.25, A 0, B 90, C 0, E1 0, E2 0, E3 0, E4 0} C_DIS
LIN {X 76.497, Y 94.755, Z 268.25, A 0, B 90, C 0, E1 0, E2 0, E3 0, E4 0} C_DIS
LIN {X 78.799, Y 91.368, Z 268.25, A 0, B 90, C 0, E1 0, E2 0, E3 0, E4 0} C_DIS
LIN {X 80.639, Y 87.708, Z 268.25, A 0, B 90, C 0, E1 0, E2 0, E3 0, E4 0} C_DIS
LIN {X 82.113, Y 83.885, Z 268.25, A 0, B 90, C 0, E1 0, E2 0, E3 0, E4 0} C_DIS
LIN {X 83.313, Y 79.966, Z 268.25, A 0, B 90, C 0, E1 0, E2 0, E3 0, E4 0} C_DIS
LIN {X 84.33, Y 75.996, Z 268.25, A 0, B 90, C 0, E1 0, E2 0, E3 0, E4 0} C_DIS
LIN {X 85.266, Y 72.005, Z 268.25, A 0, B 90, C 0, E1 0, E2 0, E3 0, E4 0} C_DIS
LIN {X 86.253, Y 68.027, Z 268.25, A 0, B 90, C 0, E1 0, E2 0, E3 0, E4 0} C_DIS
LIN {X 87.492, Y 64.122, Z 268.25, A 0, B 90, C 0, E1 0, E2 0, E3 0, E4 0} C_DIS
LIN {X 89.286, Y 60.444, Z 268.25, A 0, B 90, C 0, E1 0, E2 0, E3 0, E4 0} C_DIS
LIN {X 91.864, Y 57.271, Z 268.25, A 0, B 90, C 0, E1 0, E2 0, E3 0, E4 0} C_DIS
LIN {X 95.059, Y 54.711, Z 268.25, A 0, B 90, C 0, E1 0, E2 0, E3 0, E4 0} C_DIS
LIN {X 98.544, Y 52.556, Z 268.25, A 0, B 90, C 0, E1 0, E2 0, E3 0, E4 0} C_DIS
LIN {X 102.127, Y 50.565, Z 268.25, A 0, B 90, C 0, E1 0, E2 0, E3 0, E4 0} C_DIS
LIN {X 105.714, Y 48.582, Z 268.25, A 0, B 90, C 0, E1 0, E2 0, E3 0, E4 0} C_DIS
LIN {X 109.248, Y 46.505, Z 268.25, A 0, B 90, C 0, E1 0, E2 0, E3 0, E4 0} C_DIS
LIN {X 112.678, Y 44.262, Z 268.25, A 0, B 90, C 0, E1 0, E2 0, E3 0, E4 0} C_DIS
LIN {X 115.948, Y 41.794, Z 268.25, A 0, B 90, C 0, E1 0, E2 0, E3 0, E4 0} C_DIS
LIN {X 118.988, Y 39.046, Z 268.25, A 0, B 90, C 0, E1 0, E2 0, E3 0, E4 0} C_DIS
LIN {X 121.694, Y 35.972, Z 268.25, A 0, B 90, C 0, E1 0, E2 0, E3 0, E4 0} C_DIS
LIN {X 123.922, Y 32.536, Z 268.25, A 0, B 90, C 0, E1 0, E2 0, E3 0, E4 0} C_DIS
LIN {X 125.482, Y 28.754, Z 268.25, A 0, B 90, C 0, E1 0, E2 0, E3 0, E4 0} C_DIS
LIN {X 126.196, Y 24.726, Z 268.25, A 0, B 90, C 0, E1 0, E2 0, E3 0, E4 0} C_DIS
LIN {X 126.002, Y 20.64, Z 268.25, A 0, B 90, C 0, E1 0, E2 0, E3 0, E4 0} C_DIS
LIN {X 125.001, Y 16.671, Z 268.25, A 0, B 90, C 0, E1 0, E2 0, E3 0, E4 0} C_DIS
LIN {X 123.375, Y 12.912, Z 268.25, A 0, B 90, C 0, E1 0, E2 0, E3 0, E4 0} C_DIS
LIN {X 121.297, Y 9.382, Z 268.25, A 0, B 90, C 0, E1 0, E2 0, E3 0, E4 0} C_DIS
LIN {X 118.893, Y 6.063, Z 268.25, A 0, B 90, C 0, E1 0, E2 0, E3 0, E4 0} C_DIS
LIN {X 116.25, Y 2.934, Z 268.25, A 0, B 90, C 0, E1 0, E2 0, E3 0, E4 0} C_DIS
LIN {X 113.532, Y 0, Z 268.25, A 0, B 90, C 0, E1 0, E2 0, E3 0, E4 0} C_DIS
LIN {X 110.633, Y -2.58, Z 268.25, A 0, B 90, C 0, E1 0, E2 0, E3 0, E4 0} C_DIS
LIN {X 107.706, Y -5.447, Z 268.25, A 0, B 90, C 0, E1 0, E2 0, E3 0, E4 0} C_DIS
LIN {X 104.801, Y -8.339, Z 268.25, A 0, B 90, C 0, E1 0, E2 0, E3 0, E4 0} C_DIS
LIN {X 101.995, Y -11.326, Z 268.25, A 0, B 90, C 0, E1 0, E2 0, E3 0, E4 0} C_DIS
LIN {X 99.46, Y -14.543, Z 268.25, A 0, B 90, C 0, E1 0, E2 0, E3 0, E4 0} C_DIS
LIN {X 97.535, Y -18.152, Z 268.25, A 0, B 90, C 0, E1 0, E2 0, E3 0, E4 0} C_DIS
LIN {X 96.601, Y -22.13, Z 268.25, A 0, B 90, C 0, E1 0, E2 0, E3 0, E4 0} C_DIS
LIN {X 96.601, Y -26.223, Z 268.25, A 0, B 90, C 0, E1 0, E2 0, E3 0, E4 0} C_DIS
LIN {X 97.155, Y -30.283, Z 268.25, A 0, B 90, C 0, E1 0, E2 0, E3 0, E4 0} C_DIS
LIN {X 97.983, Y -34.297, Z 268.25, A 0, B 90, C 0, E1 0, E2 0, E3 0, E4 0} C_DIS
LIN {X 98.933, Y -38.284, Z 268.25, A 0, B 90, C 0, E1 0, E2 0, E3 0, E4 0} C_DIS
LIN {X 99.915, Y -42.263, Z 268.25, A 0, B 90, C 0, E1 0, E2 0, E3 0, E4 0} C_DIS
LIN {X 100.854, Y -46.253, Z 268.25, A 0, B 90, C 0, E1 0, E2 0, E3 0, E4 0} C_DIS
LIN {X 101.675, Y -50.268, Z 268.25, A 0, B 90, C 0, E1 0, E2 0, E3 0, E4 0} C_DIS
LIN {X 102.285, Y -54.321, Z 268.25, A 0, B 90, C 0, E1 0, E2 0, E3 0, E4 0} C_DIS
LIN {X 102.572, Y -58.408, Z 268.25, A 0, B 90, C 0, E1 0, E2 0, E3 0, E4 0} C_DIS
LIN {X 102.395, Y -62.5, Z 268.25, A 0, B 90, C 0, E1 0, E2 0, E3 0, E4 0} C_DIS
LIN {X 101.592, Y -66.514, Z 268.25, A 0, B 90, C 0, E1 0, E2 0, E3 0, E4 0} C_DIS
LIN {X 100.033, Y -70.297, Z 268.25, A 0, B 90, C 0, E1 0, E2 0, E3 0, E4 0} C_DIS
LIN {X 97.708, Y -73.663, Z 268.25, A 0, B 90, C 0, E1 0, E2 0, E3 0, E4 0} C_DIS
LIN {X 94.755, Y -76.497, Z 268.25, A 0, B 90, C 0, E1 0, E2 0, E3 0, E4 0} C_DIS
LIN {X 91.368, Y -78.799, Z 268.25, A 0, B 90, C 0, E1 0, E2 0, E3 0, E4 0} C_DIS
LIN {X 87.708, Y -80.639, Z 268.25, A 0, B 90, C 0, E1 0, E2 0, E3 0, E4 0} C_DIS
LIN {X 83.885, Y -82.113, Z 268.25, A 0, B 90, C 0, E1 0, E2 0, E3 0, E4 0} C_DIS
LIN {X 79.966, Y -83.313, Z 268.25, A 0, B 90, C 0, E1 0, E2 0, E3 0, E4 0} C_DIS
LIN {X 75.996, Y -84.33, Z 268.25, A 0, B 90, C 0, E1 0, E2 0, E3 0, E4 0} C_DIS
LIN {X 72.005, Y -85.266, Z 268.25, A 0, B 90, C 0, E1 0, E2 0, E3 0, E4 0} C_DIS
LIN {X 68.027, Y -86.253, Z 268.25, A 0, B 90, C 0, E1 0, E2 0, E3 0, E4 0} C_DIS
LIN {X 64.122, Y -87.492, Z 268.25, A 0, B 90, C 0, E1 0, E2 0, E3 0, E4 0} C_DIS
LIN {X 60.444, Y -89.286, Z 268.25, A 0, B 90, C 0, E1 0, E2 0, E3 0, E4 0} C_DIS
LIN {X 57.271, Y -91.864, Z 268.25, A 0, B 90, C 0, E1 0, E2 0, E3 0, E4 0} C_DIS
LIN {X 54.711, Y -95.059, Z 268.25, A 0, B 90, C 0, E1 0, E2 0, E3 0, E4 0} C_DIS
LIN {X 52.556, Y -98.544, Z 268.25, A 0, B 90, C 0, E1 0, E2 0, E3 0, E4 0} C_DIS
LIN {X 50.565, Y -102.127, Z 268.25, A 0, B 90, C 0, E1 0, E2 0, E3 0, E4 0} C_DIS
LIN {X 48.582, Y -105.714, Z 268.25, A 0, B 90, C 0, E1 0, E2 0, E3 0, E4 0} C_DIS
LIN {X 46.505, Y -109.248, Z 268.25, A 0, B 90, C 0, E1 0, E2 0, E3 0, E4 0} C_DIS
LIN {X 44.262, Y -112.678, Z 268.25, A 0, B 90, C 0, E1 0, E2 0, E3 0, E4 0} C_DIS
LIN {X 41.794, Y -115.948, Z 268.25, A 0, B 90, C 0, E1 0, E2 0, E3 0, E4 0} C_DIS
LIN {X 39.046, Y -118.988, Z 268.25, A 0, B 90, C 0, E1 0, E2 0, E3 0, E4 0} C_DIS
LIN {X 35.972, Y -121.694, Z 268.25, A 0, B 90, C 0, E1 0, E2 0, E3 0, E4 0} C_DIS
LIN {X 32.536, Y -123.922, Z 268.25, A 0, B 90, C 0, E1 0, E2 0, E3 0, E4 0} C_DIS
LIN {X 28.754, Y -125.482, Z 268.25, A 0, B 90, C 0, E1 0, E2 0, E3 0, E4 0} C_DIS
LIN {X 24.726, Y -126.196, Z 268.25, A 0, B 90, C 0, E1 0, E2 0, E3 0, E4 0} C_DIS
LIN {X 20.64, Y -126.002, Z 268.25, A 0, B 90, C 0, E1 0, E2 0, E3 0, E4 0} C_DIS
LIN {X 16.671, Y -125.001, Z 268.25, A 0, B 90, C 0, E1 0, E2 0, E3 0, E4 0} C_DIS
LIN {X 12.912, Y -123.375, Z 268.25, A 0, B 90, C 0, E1 0, E2 0, E3 0, E4 0} C_DIS
LIN {X 9.382, Y -121.297, Z 268.25, A 0, B 90, C 0, E1 0, E2 0, E3 0, E4 0} C_DIS
LIN {X 6.063, Y -118.893, Z 268.25, A 0, B 90, C 0, E1 0, E2 0, E3 0, E4 0} C_DIS
LIN {X 2.934, Y -116.25, Z 268.25, A 0, B 90, C 0, E1 0, E2 0, E3 0, E4 0} C_DIS
LIN {X 0, Y -113.532, Z 268.25, A 0, B 90, C 0, E1 0, E2 0, E3 0, E4 0} C_DIS
LIN {X -2.58, Y -110.633, Z 268.25, A 0, B 90, C 0, E1 0, E2 0, E3 0, E4 0} C_DIS
LIN {X -5.447, Y -107.706, Z 268.25, A 0, B 90, C 0, E1 0, E2 0, E3 0, E4 0} C_DIS
LIN {X -8.339, Y -104.801, Z 268.25, A 0, B 90, C 0, E1 0, E2 0, E3 0, E4 0} C_DIS
LIN {X -11.326, Y -101.995, Z 268.25, A 0, B 90, C 0, E1 0, E2 0, E3 0, E4 0} C_DIS
LIN {X -14.543, Y -99.46, Z 268.25, A 0, B 90, C 0, E1 0, E2 0, E3 0, E4 0} C_DIS
LIN {X -18.152, Y -97.535, Z 268.25, A 0, B 90, C 0, E1 0, E2 0, E3 0, E4 0} C_DIS
LIN {X -22.13, Y -96.601, Z 268.25, A 0, B 90, C 0, E1 0, E2 0, E3 0, E4 0} C_DIS
LIN {X -26.223, Y -96.601, Z 268.25, A 0, B 90, C 0, E1 0, E2 0, E3 0, E4 0} C_DIS
LIN {X -30.283, Y -97.155, Z 268.25, A 0, B 90, C 0, E1 0, E2 0, E3 0, E4 0} C_DIS
LIN {X -34.297, Y -97.983, Z 268.25, A 0, B 90, C 0, E1 0, E2 0, E3 0, E4 0} C_DIS
LIN {X -38.284, Y -98.933, Z 268.25, A 0, B 90, C 0, E1 0, E2 0, E3 0, E4 0} C_DIS
LIN {X -42.263, Y -99.915, Z 268.25, A 0, B 90, C 0, E1 0, E2 0, E3 0, E4 0} C_DIS
LIN {X -46.253, Y -100.854, Z 268.25, A 0, B 90, C 0, E1 0, E2 0, E3 0, E4 0} C_DIS
LIN {X -50.268, Y -101.675, Z 268.25, A 0, B 90, C 0, E1 0, E2 0, E3 0, E4 0} C_DIS
LIN {X -54.321, Y -102.285, Z 268.25, A 0, B 90, C 0, E1 0, E2 0, E3 0, E4 0} C_DIS
LIN {X -58.408, Y -102.572, Z 268.25, A 0, B 90, C 0, E1 0, E2 0, E3 0, E4 0} C_DIS
LIN {X -62.5, Y -102.395, Z 268.25, A 0, B 90, C 0, E1 0, E2 0, E3 0, E4 0} C_DIS
LIN {X -66.514, Y -101.592, Z 268.25, A 0, B 90, C 0, E1 0, E2 0, E3 0, E4 0} C_DIS
LIN {X -70.297, Y -100.033, Z 268.25, A 0, B 90, C 0, E1 0, E2 0, E3 0, E4 0} C_DIS
LIN {X -73.663, Y -97.708, Z 268.25, A 0, B 90, C 0, E1 0, E2 0, E3 0, E4 0} C_DIS
LIN {X -76.497, Y -94.755, Z 268.25, A 0, B 90, C 0, E1 0, E2 0, E3 0, E4 0} C_DIS
LIN {X -78.799, Y -91.368, Z 268.25, A 0, B 90, C 0, E1 0, E2 0, E3 0, E4 0} C_DIS
LIN {X -80.639, Y -87.708, Z 268.25, A 0, B 90, C 0, E1 0, E2 0, E3 0, E4 0} C_DIS
LIN {X -82.113, Y -83.885, Z 268.25, A 0, B 90, C 0, E1 0, E2 0, E3 0, E4 0} C_DIS
LIN {X -83.313, Y -79.966, Z 268.25, A 0, B 90, C 0, E1 0, E2 0, E3 0, E4 0} C_DIS
LIN {X -84.33, Y -75.996, Z 268.25, A 0, B 90, C 0, E1 0, E2 0, E3 0, E4 0} C_DIS
LIN {X -85.266, Y -72.005, Z 268.25, A 0, B 90, C 0, E1 0, E2 0, E3 0, E4 0} C_DIS
LIN {X -86.253, Y -68.027, Z 268.25, A 0, B 90, C 0, E1 0, E2 0, E3 0, E4 0} C_DIS
LIN {X -87.492, Y -64.122, Z 268.25, A 0, B 90, C 0, E1 0, E2 0, E3 0, E4 0} C_DIS
LIN {X -89.286, Y -60.444, Z 268.25, A 0, B 90, C 0, E1 0, E2 0, E3 0, E4 0} C_DIS
LIN {X -91.864, Y -57.271, Z 268.25, A 0, B 90, C 0, E1 0, E2 0, E3 0, E4 0} C_DIS
LIN {X -95.059, Y -54.711, Z 268.25, A 0, B 90, C 0, E1 0, E2 0, E3 0, E4 0} C_DIS
LIN {X -98.544, Y -52.556, Z 268.25, A 0, B 90, C 0, E1 0, E2 0, E3 0, E4 0} C_DIS
LIN {X -102.127, Y -50.565, Z 268.25, A 0, B 90, C 0, E1 0, E2 0, E3 0, E4 0} C_DIS
LIN {X -105.714, Y -48.582, Z 268.25, A 0, B 90, C 0, E1 0, E2 0, E3 0, E4 0} C_DIS
LIN {X -109.248, Y -46.505, Z 268.25, A 0, B 90, C 0, E1 0, E2 0, E3 0, E4 0} C_DIS
LIN {X -112.678, Y -44.262, Z 268.25, A 0, B 90, C 0, E1 0, E2 0, E3 0, E4 0} C_DIS
LIN {X -115.948, Y -41.794, Z 268.25, A 0, B 90, C 0, E1 0, E2 0, E3 0, E4 0} C_DIS
LIN {X -118.988, Y -39.046, Z 268.25, A 0, B 90, C 0, E1 0, E2 0, E3 0, E4 0} C_DIS
LIN {X -121.694, Y -35.972, Z 268.25, A 0, B 90, C 0, E1 0, E2 0, E3 0, E4 0} C_DIS
LIN {X -123.922, Y -32.536, Z 268.25, A 0, B 90, C 0, E1 0, E2 0, E3 0, E4 0} C_DIS
LIN {X -125.482, Y -28.754, Z 268.25, A 0, B 90, C 0, E1 0, E2 0, E3 0, E4 0} C_DIS
LIN {X -126.196, Y -24.726, Z 268.25, A 0, B 90, C 0, E1 0, E2 0, E3 0, E4 0} C_DIS
LIN {X -126.002, Y -20.64, Z 268.25, A 0, B 90, C 0, E1 0, E2 0, E3 0, E4 0} C_DIS
LIN {X -125.001, Y -16.671, Z 268.25, A 0, B 90, C 0, E1 0, E2 0, E3 0, E4 0} C_DIS
LIN {X -123.375, Y -12.912, Z 268.25, A 0, B 90, C 0, E1 0, E2 0, E3 0, E4 0} C_DIS
LIN {X -121.297, Y -9.382, Z 268.25, A 0, B 90, C 0, E1 0, E2 0, E3 0, E4 0} C_DIS
LIN {X -118.893, Y -6.063, Z 268.25, A 0, B 90, C 0, E1 0, E2 0, E3 0, E4 0} C_DIS
LIN {X -116.25, Y -2.934, Z 268.25, A 0, B 90, C 0, E1 0, E2 0, E3 0, E4 0} C_DIS
LIN {X -114.376, Y 0, Z 270.75, A 0, B 90, C 0, E1 0, E2 0, E3 0, E4 0} C_DIS
LIN {X -111.44, Y 2.611, Z 270.75, A 0, B 90, C 0, E1 0, E2 0, E3 0, E4 0} C_DIS
LIN {X -108.472, Y 5.504, Z 270.75, A 0, B 90, C 0, E1 0, E2 0, E3 0, E4 0} C_DIS
LIN {X -105.529, Y 8.424, Z 270.75, A 0, B 90, C 0, E1 0, E2 0, E3 0, E4 0} C_DIS
LIN {X -102.691, Y 11.445, Z 270.75, A 0, B 90, C 0, E1 0, E2 0, E3 0, E4 0} C_DIS
LIN {X -100.139, Y 14.708, Z 270.75, A 0, B 90, C 0, E1 0, E2 0, E3 0, E4 0} C_DIS
LIN {X -98.228, Y 18.376, Z 270.75, A 0, B 90, C 0, E1 0, E2 0, E3 0, E4 0} C_DIS
LIN {X -97.349, Y 22.414, Z 270.75, A 0, B 90, C 0, E1 0, E2 0, E3 0, E4 0} C_DIS
LIN {X -97.429, Y 26.553, Z 270.75, A 0, B 90, C 0, E1 0, E2 0, E3 0, E4 0} C_DIS
LIN {X -98.068, Y 30.647, Z 270.75, A 0, B 90, C 0, E1 0, E2 0, E3 0, E4 0} C_DIS
LIN {X -98.979, Y 34.691, Z 270.75, A 0, B 90, C 0, E1 0, E2 0, E3 0, E4 0} C_DIS
LIN {X -100.005, Y 38.708, Z 270.75, A 0, B 90, C 0, E1 0, E2 0, E3 0, E4 0} C_DIS
LIN {X -101.052, Y 42.719, Z 270.75, A 0, B 90, C 0, E1 0, E2 0, E3 0, E4 0} C_DIS
LIN {X -102.046, Y 46.743, Z 270.75, A 0, B 90, C 0, E1 0, E2 0, E3 0, E4 0} C_DIS
LIN {X -102.908, Y 50.798, Z 270.75, A 0, B 90, C 0, E1 0, E2 0, E3 0, E4 0} C_DIS
LIN {X -103.545, Y 54.894, Z 270.75, A 0, B 90, C 0, E1 0, E2 0, E3 0, E4 0} C_DIS
LIN {X -103.84, Y 59.027, Z 270.75, A 0, B 90, C 0, E1 0, E2 0, E3 0, E4 0} C_DIS
LIN {X -103.648, Y 63.165, Z 270.75, A 0, B 90, C 0, E1 0, E2 0, E3 0, E4 0} C_DIS
LIN {X -102.803, Y 67.218, Z 270.75, A 0, B 90, C 0, E1 0, E2 0, E3 0, E4 0} C_DIS
LIN {X -101.174, Y 71.021, Z 270.75, A 0, B 90, C 0, E1 0, E2 0, E3 0, E4 0} C_DIS
LIN {X -98.76, Y 74.381, Z 270.75, A 0, B 90, C 0, E1 0, E2 0, E3 0, E4 0} C_DIS
LIN {X -95.712, Y 77.182, Z 270.75, A 0, B 90, C 0, E1 0, E2 0, E3 0, E4 0} C_DIS
LIN {X -92.233, Y 79.428, Z 270.75, A 0, B 90, C 0, E1 0, E2 0, E3 0, E4 0} C_DIS
LIN {X -88.487, Y 81.201, Z 270.75, A 0, B 90, C 0, E1 0, E2 0, E3 0, E4 0} C_DIS
LIN {X -84.586, Y 82.598, Z 270.75, A 0, B 90, C 0, E1 0, E2 0, E3 0, E4 0} C_DIS
LIN {X -80.595, Y 83.717, Z 270.75, A 0, B 90, C 0, E1 0, E2 0, E3 0, E4 0} C_DIS
LIN {X -76.556, Y 84.653, Z 270.75, A 0, B 90, C 0, E1 0, E2 0, E3 0, E4 0} C_DIS
LIN {X -72.5, Y 85.508, Z 270.75, A 0, B 90, C 0, E1 0, E2 0, E3 0, E4 0} C_DIS
LIN {X -68.456, Y 86.42, Z 270.75, A 0, B 90, C 0, E1 0, E2 0, E3 0, E4 0} C_DIS
LIN {X -64.482, Y 87.594, Z 270.75, A 0, B 90, C 0, E1 0, E2 0, E3 0, E4 0} C_DIS
LIN {X -60.731, Y 89.341, Z 270.75, A 0, B 90, C 0, E1 0, E2 0, E3 0, E4 0} C_DIS
LIN {X -57.491, Y 91.91, Z 270.75, A 0, B 90, C 0, E1 0, E2 0, E3 0, E4 0} C_DIS
LIN {X -54.893, Y 95.134, Z 270.75, A 0, B 90, C 0, E1 0, E2 0, E3 0, E4 0} C_DIS
LIN {X -52.729, Y 98.668, Z 270.75, A 0, B 90, C 0, E1 0, E2 0, E3 0, E4 0} C_DIS
LIN {X -50.747, Y 102.309, Z 270.75, A 0, B 90, C 0, E1 0, E2 0, E3 0, E4 0} C_DIS
LIN {X -48.784, Y 105.96, Z 270.75, A 0, B 90, C 0, E1 0, E2 0, E3 0, E4 0} C_DIS
LIN {X -46.734, Y 109.563, Z 270.75, A 0, B 90, C 0, E1 0, E2 0, E3 0, E4 0} C_DIS
LIN {X -44.521, Y 113.068, Z 270.75, A 0, B 90, C 0, E1 0, E2 0, E3 0, E4 0} C_DIS
LIN {X -42.082, Y 116.419, Z 270.75, A 0, B 90, C 0, E1 0, E2 0, E3 0, E4 0} C_DIS
LIN {X -39.361, Y 119.544, Z 270.75, A 0, B 90, C 0, E1 0, E2 0, E3 0, E4 0} C_DIS
LIN {X -36.305, Y 122.341, Z 270.75, A 0, B 90, C 0, E1 0, E2 0, E3 0, E4 0} C_DIS
LIN {X -32.875, Y 124.661, Z 270.75, A 0, B 90, C 0, E1 0, E2 0, E3 0, E4 0} C_DIS
LIN {X -29.079, Y 126.31, Z 270.75, A 0, B 90, C 0, E1 0, E2 0, E3 0, E4 0} C_DIS
LIN {X -25.018, Y 127.097, Z 270.75, A 0, B 90, C 0, E1 0, E2 0, E3 0, E4 0} C_DIS
LIN {X -20.884, Y 126.95, Z 270.75, A 0, B 90, C 0, E1 0, E2 0, E3 0, E4 0} C_DIS
LIN {X -16.862, Y 125.967, Z 270.75, A 0, B 90, C 0, E1 0, E2 0, E3 0, E4 0} C_DIS
LIN {X -13.054, Y 124.338, Z 270.75, A 0, B 90, C 0, E1 0, E2 0, E3 0, E4 0} C_DIS
LIN {X -9.48, Y 122.242, Z 270.75, A 0, B 90, C 0, E1 0, E2 0, E3 0, E4 0} C_DIS
LIN {X -6.125, Y 119.81, Z 270.75, A 0, B 90, C 0, E1 0, E2 0, E3 0, E4 0} C_DIS
LIN {X -2.962, Y 117.133, Z 270.75, A 0, B 90, C 0, E1 0, E2 0, E3 0, E4 0} C_DIS
LIN {X 0, Y 114.376, Z 270.75, A 0, B 90, C 0, E1 0, E2 0, E3 0, E4 0} C_DIS
LIN {X 2.611, Y 111.44, Z 270.75, A 0, B 90, C 0, E1 0, E2 0, E3 0, E4 0} C_DIS
LIN {X 5.504, Y 108.472, Z 270.75, A 0, B 90, C 0, E1 0, E2 0, E3 0, E4 0} C_DIS
LIN {X 8.424, Y 105.529, Z 270.75, A 0, B 90, C 0, E1 0, E2 0, E3 0, E4 0} C_DIS
LIN {X 11.445, Y 102.691, Z 270.75, A 0, B 90, C 0, E1 0, E2 0, E3 0, E4 0} C_DIS
LIN {X 14.708, Y 100.139, Z 270.75, A 0, B 90, C 0, E1 0, E2 0, E3 0, E4 0} C_DIS
LIN {X 18.376, Y 98.228, Z 270.75, A 0, B 90, C 0, E1 0, E2 0, E3 0, E4 0} C_DIS
LIN {X 22.414, Y 97.349, Z 270.75, A 0, B 90, C 0, E1 0, E2 0, E3 0, E4 0} C_DIS
LIN {X 26.553, Y 97.429, Z 270.75, A 0, B 90, C 0, E1 0, E2 0, E3 0, E4 0} C_DIS
LIN {X 30.647, Y 98.068, Z 270.75, A 0, B 90, C 0, E1 0, E2 0, E3 0, E4 0} C_DIS
LIN {X 34.691, Y 98.979, Z 270.75, A 0, B 90, C 0, E1 0, E2 0, E3 0, E4 0} C_DIS
LIN {X 38.708, Y 100.005, Z 270.75, A 0, B 90, C 0, E1 0, E2 0, E3 0, E4 0} C_DIS
LIN {X 42.719, Y 101.052, Z 270.75, A 0, B 90, C 0, E1 0, E2 0, E3 0, E4 0} C_DIS
LIN {X 46.743, Y 102.046, Z 270.75, A 0, B 90, C 0, E1 0, E2 0, E3 0, E4 0} C_DIS
LIN {X 50.798, Y 102.908, Z 270.75, A 0, B 90, C 0, E1 0, E2 0, E3 0, E4 0} C_DIS
LIN {X 54.894, Y 103.545, Z 270.75, A 0, B 90, C 0, E1 0, E2 0, E3 0, E4 0} C_DIS
LIN {X 59.027, Y 103.84, Z 270.75, A 0, B 90, C 0, E1 0, E2 0, E3 0, E4 0} C_DIS
LIN {X 63.165, Y 103.648, Z 270.75, A 0, B 90, C 0, E1 0, E2 0, E3 0, E4 0} C_DIS
LIN {X 67.218, Y 102.803, Z 270.75, A 0, B 90, C 0, E1 0, E2 0, E3 0, E4 0} C_DIS
LIN {X 71.021, Y 101.174, Z 270.75, A 0, B 90, C 0, E1 0, E2 0, E3 0, E4 0} C_DIS
LIN {X 74.381, Y 98.76, Z 270.75, A 0, B 90, C 0, E1 0, E2 0, E3 0, E4 0} C_DIS
LIN {X 77.182, Y 95.712, Z 270.75, A 0, B 90, C 0, E1 0, E2 0, E3 0, E4 0} C_DIS
LIN {X 79.428, Y 92.233, Z 270.75, A 0, B 90, C 0, E1 0, E2 0, E3 0, E4 0} C_DIS
LIN {X 81.201, Y 88.487, Z 270.75, A 0, B 90, C 0, E1 0, E2 0, E3 0, E4 0} C_DIS
LIN {X 82.598, Y 84.586, Z 270.75, A 0, B 90, C 0, E1 0, E2 0, E3 0, E4 0} C_DIS
LIN {X 83.717, Y 80.595, Z 270.75, A 0, B 90, C 0, E1 0, E2 0, E3 0, E4 0} C_DIS
LIN {X 84.653, Y 76.556, Z 270.75, A 0, B 90, C 0, E1 0, E2 0, E3 0, E4 0} C_DIS
LIN {X 85.508, Y 72.5, Z 270.75, A 0, B 90, C 0, E1 0, E2 0, E3 0, E4 0} C_DIS
LIN {X 86.42, Y 68.456, Z 270.75, A 0, B 90, C 0, E1 0, E2 0, E3 0, E4 0} C_DIS
LIN {X 87.594, Y 64.482, Z 270.75, A 0, B 90, C 0, E1 0, E2 0, E3 0, E4 0} C_DIS
LIN {X 89.341, Y 60.731, Z 270.75, A 0, B 90, C 0, E1 0, E2 0, E3 0, E4 0} C_DIS
LIN {X 91.91, Y 57.491, Z 270.75, A 0, B 90, C 0, E1 0, E2 0, E3 0, E4 0} C_DIS
LIN {X 95.134, Y 54.893, Z 270.75, A 0, B 90, C 0, E1 0, E2 0, E3 0, E4 0} C_DIS
LIN {X 98.668, Y 52.729, Z 270.75, A 0, B 90, C 0, E1 0, E2 0, E3 0, E4 0} C_DIS
LIN {X 102.309, Y 50.747, Z 270.75, A 0, B 90, C 0, E1 0, E2 0, E3 0, E4 0} C_DIS
LIN {X 105.96, Y 48.784, Z 270.75, A 0, B 90, C 0, E1 0, E2 0, E3 0, E4 0} C_DIS
LIN {X 109.563, Y 46.734, Z 270.75, A 0, B 90, C 0, E1 0, E2 0, E3 0, E4 0} C_DIS
LIN {X 113.068, Y 44.521, Z 270.75, A 0, B 90, C 0, E1 0, E2 0, E3 0, E4 0} C_DIS
